    movel([0.080813, -1.351716, -2.594300, -0.766373, 1.570796, 1.651610],accel_mss,speed_ms,0,blend_radius_m)
    movel([0.080675, -1.351545, -2.594414, -0.766430, 1.570796, 1.651471],accel_mss,speed_ms,0,blend_radius_m)
    movel([0.080768, -1.351204, -2.594640, -0.766545, 1.570796, 1.651564],accel_mss,speed_ms,0,blend_radius_m)
    movel([0.080890, -1.350900, -2.594842, -0.766647, 1.570796, 1.651686],accel_mss,speed_ms,0,blend_radius_m)
    movel([0.080645, -1.350707, -2.594969, -0.766712, 1.570796, 1.651441],accel_mss,speed_ms,0,blend_radius_m)
    movel([0.080619, -1.350492, -2.595112, -0.766785, 1.570796, 1.651416],accel_mss,speed_ms,0,blend_radius_m)
    movel([0.080919, -1.350160, -2.595332, -0.766897, 1.570796, 1.651715],accel_mss,speed_ms,0,blend_radius_m)
    movel([0.080769, -1.349809, -2.595564, -0.767016, 1.570796, 1.651566],accel_mss,speed_ms,0,blend_radius_m)
    movel([0.080640, -1.349621, -2.595688, -0.767080, 1.570796, 1.651436],accel_mss,speed_ms,0,blend_radius_m)
    movel([0.080628, -1.349397, -2.595836, -0.767155, 1.570796, 1.651424],accel_mss,speed_ms,0,blend_radius_m)
    movel([0.080942, -1.348990, -2.596105, -0.767294, 1.570796, 1.651739],accel_mss,speed_ms,0,blend_radius_m)
    movel([0.081368, -1.348809, -2.596225, -0.767355, 1.570796, 1.652164],accel_mss,speed_ms,0,blend_radius_m)
    movel([0.083131, -1.348413, -2.596486, -0.767490, 1.570796, 1.653928],accel_mss,speed_ms,0,blend_radius_m)
    speed_ms = 0.003
    movel([0.083131, -1.335017, -2.590258, -0.787114, 1.570796, 1.653928],accel_mss,speed_ms,0,blend_radius_m)
    speed_ms = 1.000
    movel([0.083131, -1.309400, -2.577409, -0.825580, 1.570796, 1.653928],accel_mss,speed_ms,0,blend_radius_m)
    movel([0.082638, -1.312886, -2.575230, -0.824273, 1.570796, 1.653435],accel_mss,speed_ms,0,blend_radius_m)
    movel([0.082638, -1.338446, -2.588033, -0.785910, 1.570796, 1.653435],accel_mss,speed_ms,0,blend_radius_m)
    speed_ms = 0.003
    movel([0.082638, -1.348431, -2.592700, -0.771258, 1.570796, 1.653435],accel_mss,speed_ms,0,blend_radius_m)
    speed_ms = 0.007
    movel([0.083010, -1.348325, -2.592770, -0.771294, 1.570796, 1.653806],accel_mss,speed_ms,0,blend_radius_m)
    movel([0.083255, -1.348397, -2.592722, -0.771269, 1.570796, 1.654051],accel_mss,speed_ms,0,blend_radius_m)
    movel([0.083272, -1.348613, -2.592580, -0.771196, 1.570796, 1.654068],accel_mss,speed_ms,0,blend_radius_m)
    movel([0.082991, -1.348882, -2.592402, -0.771105, 1.570796, 1.653788],accel_mss,speed_ms,0,blend_radius_m)
    movel([0.082561, -1.349059, -2.592285, -0.771045, 1.570796, 1.653357],accel_mss,speed_ms,0,blend_radius_m)
    movel([0.082329, -1.349028, -2.592305, -0.771056, 1.570796, 1.653125],accel_mss,speed_ms,0,blend_radius_m)
    movel([0.082337, -1.348676, -2.592538, -0.771175, 1.570796, 1.653134],accel_mss,speed_ms,0,blend_radius_m)
    movel([0.082638, -1.348431, -2.592700, -0.771258, 1.570796, 1.653435],accel_mss,speed_ms,0,blend_radius_m)
    speed_ms = 0.003
    movel([0.082638, -1.351808, -2.594239, -0.766342, 1.570796, 1.653435],accel_mss,speed_ms,0,blend_radius_m)
    speed_ms = 0.007
    movel([0.083010, -1.351702, -2.594309, -0.766377, 1.570796, 1.653806],accel_mss,speed_ms,0,blend_radius_m)
    movel([0.083255, -1.351775, -2.594261, -0.766353, 1.570796, 1.654051],accel_mss,speed_ms,0,blend_radius_m)
    movel([0.083272, -1.351990, -2.594118, -0.766281, 1.570796, 1.654068],accel_mss,speed_ms,0,blend_radius_m)
    movel([0.082991, -1.352258, -2.593940, -0.766191, 1.570796, 1.653788],accel_mss,speed_ms,0,blend_radius_m)
    movel([0.082561, -1.352435, -2.593823, -0.766132, 1.570796, 1.653357],accel_mss,speed_ms,0,blend_radius_m)
    movel([0.082329, -1.352404, -2.593843, -0.766142, 1.570796, 1.653125],accel_mss,speed_ms,0,blend_radius_m)
    movel([0.082337, -1.352052, -2.594077, -0.766260, 1.570796, 1.653134],accel_mss,speed_ms,0,blend_radius_m)
    movel([0.082638, -1.351808, -2.594239, -0.766342, 1.570796, 1.653435],accel_mss,speed_ms,0,blend_radius_m)
    speed_ms = 0.003
    movel([0.082638, -1.338446, -2.588033, -0.785910, 1.570796, 1.653435],accel_mss,speed_ms,0,blend_radius_m)
    speed_ms = 1.000
    movel([0.082638, -1.312886, -2.575230, -0.824273, 1.570796, 1.653435],accel_mss,speed_ms,0,blend_radius_m)
    movel([0.075847, -1.319560, -2.571014, -0.821815, 1.570796, 1.646643],accel_mss,speed_ms,0,blend_radius_m)
    movel([0.075847, -1.345010, -2.583731, -0.783648, 1.570796, 1.646643],accel_mss,speed_ms,0,blend_radius_m)
    speed_ms = 0.003
    movel([0.075847, -1.354947, -2.588365, -0.769077, 1.570796, 1.646643],accel_mss,speed_ms,0,blend_radius_m)
    speed_ms = 0.007
    movel([0.076210, -1.355243, -2.588167, -0.768979, 1.570796, 1.647006],accel_mss,speed_ms,0,blend_radius_m)
    movel([0.076357, -1.355481, -2.588008, -0.768901, 1.570796, 1.647154],accel_mss,speed_ms,0,blend_radius_m)
    movel([0.076398, -1.355704, -2.587858, -0.768827, 1.570796, 1.647194],accel_mss,speed_ms,0,blend_radius_m)
    movel([0.076337, -1.355959, -2.587687, -0.768743, 1.570796, 1.647134],accel_mss,speed_ms,0,blend_radius_m)
    movel([0.076172, -1.356294, -2.587462, -0.768633, 1.570796, 1.646969],accel_mss,speed_ms,0,blend_radius_m)
    movel([0.075752, -1.356855, -2.587085, -0.768449, 1.570796, 1.646548],accel_mss,speed_ms,0,blend_radius_m)
    movel([0.075239, -1.357270, -2.586806, -0.768313, 1.570796, 1.646035],accel_mss,speed_ms,0,blend_radius_m)
    movel([0.074675, -1.357502, -2.586649, -0.768238, 1.570796, 1.645471],accel_mss,speed_ms,0,blend_radius_m)
    movel([0.074114, -1.357533, -2.586628, -0.768227, 1.570796, 1.644910],accel_mss,speed_ms,0,blend_radius_m)
    movel([0.073609, -1.357253, -2.586817, -0.768319, 1.570796, 1.644405],accel_mss,speed_ms,0,blend_radius_m)
    movel([0.073464, -1.356659, -2.587216, -0.768513, 1.570796, 1.644260],accel_mss,speed_ms,0,blend_radius_m)
    movel([0.073721, -1.355938, -2.587701, -0.768750, 1.570796, 1.644518],accel_mss,speed_ms,0,blend_radius_m)
    movel([0.074305, -1.355315, -2.588118, -0.768955, 1.570796, 1.645101],accel_mss,speed_ms,0,blend_radius_m)
    movel([0.074876, -1.354985, -2.588340, -0.769064, 1.570796, 1.645673],accel_mss,speed_ms,0,blend_radius_m)
    movel([0.075398, -1.354858, -2.588425, -0.769106, 1.570796, 1.646194],accel_mss,speed_ms,0,blend_radius_m)
    movel([0.075847, -1.354947, -2.588365, -0.769077, 1.570796, 1.646643],accel_mss,speed_ms,0,blend_radius_m)
    speed_ms = 0.003
    movel([0.075847, -1.358308, -2.589893, -0.764188, 1.570796, 1.646643],accel_mss,speed_ms,0,blend_radius_m)
    speed_ms = 0.007
    movel([0.076210, -1.358603, -2.589694, -0.764092, 1.570796, 1.647006],accel_mss,speed_ms,0,blend_radius_m)
    movel([0.076357, -1.358840, -2.589535, -0.764014, 1.570796, 1.647154],accel_mss,speed_ms,0,blend_radius_m)
    movel([0.076398, -1.359063, -2.589385, -0.763942, 1.570796, 1.647194],accel_mss,speed_ms,0,blend_radius_m)
    movel([0.076337, -1.359317, -2.589213, -0.763859, 1.570796, 1.647134],accel_mss,speed_ms,0,blend_radius_m)
    movel([0.076172, -1.359651, -2.588988, -0.763751, 1.570796, 1.646969],accel_mss,speed_ms,0,blend_radius_m)
    movel([0.075752, -1.360211, -2.588610, -0.763569, 1.570796, 1.646548],accel_mss,speed_ms,0,blend_radius_m)
    movel([0.075239, -1.360624, -2.588330, -0.763435, 1.570796, 1.646035],accel_mss,speed_ms,0,blend_radius_m)
    movel([0.074675, -1.360856, -2.588173, -0.763360, 1.570796, 1.645471],accel_mss,speed_ms,0,blend_radius_m)
    movel([0.074114, -1.360887, -2.588152, -0.763350, 1.570796, 1.644910],accel_mss,speed_ms,0,blend_radius_m)
    movel([0.073609, -1.360608, -2.588341, -0.763440, 1.570796, 1.644405],accel_mss,speed_ms,0,blend_radius_m)
    movel([0.073464, -1.360015, -2.588742, -0.763632, 1.570796, 1.644260],accel_mss,speed_ms,0,blend_radius_m)
    movel([0.073721, -1.359296, -2.589227, -0.763866, 1.570796, 1.644518],accel_mss,speed_ms,0,blend_radius_m)
    movel([0.074305, -1.358675, -2.589646, -0.764068, 1.570796, 1.645101],accel_mss,speed_ms,0,blend_radius_m)
    movel([0.074876, -1.358345, -2.589868, -0.764176, 1.570796, 1.645673],accel_mss,speed_ms,0,blend_radius_m)
    movel([0.075398, -1.358219, -2.589953, -0.764217, 1.570796, 1.646194],accel_mss,speed_ms,0,blend_radius_m)
    movel([0.075847, -1.358308, -2.589893, -0.764188, 1.570796, 1.646643],accel_mss,speed_ms,0,blend_radius_m)
    speed_ms = 0.003
    movel([0.075847, -1.345010, -2.583731, -0.783648, 1.570796, 1.646643],accel_mss,speed_ms,0,blend_radius_m)
    speed_ms = 1.000
    movel([0.075847, -1.319560, -2.571014, -0.821815, 1.570796, 1.646643],accel_mss,speed_ms,0,blend_radius_m)
    movel([0.078635, -1.323961, -2.568202, -0.820226, 1.570796, 1.649431],accel_mss,speed_ms,0,blend_radius_m)
    movel([0.078635, -1.349337, -2.580862, -0.782189, 1.570796, 1.649431],accel_mss,speed_ms,0,blend_radius_m)
    speed_ms = 0.003
    movel([0.078635, -1.359242, -2.585475, -0.767671, 1.570796, 1.649431],accel_mss,speed_ms,0,blend_radius_m)
    speed_ms = 0.007
    movel([0.079474, -1.359723, -2.585151, -0.767516, 1.570796, 1.650271],accel_mss,speed_ms,0,blend_radius_m)
    movel([0.080172, -1.360238, -2.584802, -0.767349, 1.570796, 1.650969],accel_mss,speed_ms,0,blend_radius_m)
    movel([0.080222, -1.360455, -2.584655, -0.767279, 1.570796, 1.651018],accel_mss,speed_ms,0,blend_radius_m)
    movel([0.079954, -1.360655, -2.584519, -0.767215, 1.570796, 1.650750],accel_mss,speed_ms,0,blend_radius_m)
    movel([0.079275, -1.360021, -2.584949, -0.767419, 1.570796, 1.650071],accel_mss,speed_ms,0,blend_radius_m)
    movel([0.078610, -1.359377, -2.585384, -0.767628, 1.570796, 1.649406],accel_mss,speed_ms,0,blend_radius_m)
    speed_ms = 0.003
    movel([0.078635, -1.362592, -2.586996, -0.762801, 1.570796, 1.649431],accel_mss,speed_ms,0,blend_radius_m)
    speed_ms = 0.007
    movel([0.079474, -1.363071, -2.586671, -0.762648, 1.570796, 1.650271],accel_mss,speed_ms,0,blend_radius_m)
    movel([0.080172, -1.363585, -2.586321, -0.762483, 1.570796, 1.650969],accel_mss,speed_ms,0,blend_radius_m)
    movel([0.080222, -1.363801, -2.586174, -0.762414, 1.570796, 1.651018],accel_mss,speed_ms,0,blend_radius_m)
    movel([0.079954, -1.364001, -2.586038, -0.762350, 1.570796, 1.650750],accel_mss,speed_ms,0,blend_radius_m)
    movel([0.079275, -1.363368, -2.586468, -0.762552, 1.570796, 1.650071],accel_mss,speed_ms,0,blend_radius_m)
    movel([0.078610, -1.362726, -2.586905, -0.762758, 1.570796, 1.649406],accel_mss,speed_ms,0,blend_radius_m)
    speed_ms = 0.003
    movel([0.078635, -1.349337, -2.580862, -0.782189, 1.570796, 1.649431],accel_mss,speed_ms,0,blend_radius_m)
    speed_ms = 1.000
    movel([0.078635, -1.323961, -2.568202, -0.820226, 1.570796, 1.649431],accel_mss,speed_ms,0,blend_radius_m)
    movel([0.084889, -1.331749, -2.563164, -0.817476, 1.570796, 1.655685],accel_mss,speed_ms,0,blend_radius_m)
    movel([0.084889, -1.356993, -2.575725, -0.779672, 1.570796, 1.655685],accel_mss,speed_ms,0,blend_radius_m)
    speed_ms = 0.003
    movel([0.084889, -1.366841, -2.580300, -0.765248, 1.570796, 1.655685],accel_mss,speed_ms,0,blend_radius_m)
    speed_ms = 0.007
    movel([0.085264, -1.366718, -2.580384, -0.765287, 1.570796, 1.656061],accel_mss,speed_ms,0,blend_radius_m)
    movel([0.085429, -1.367001, -2.580190, -0.765198, 1.570796, 1.656225],accel_mss,speed_ms,0,blend_radius_m)
    movel([0.085290, -1.367254, -2.580016, -0.765119, 1.570796, 1.656086],accel_mss,speed_ms,0,blend_radius_m)
    movel([0.085006, -1.367407, -2.579911, -0.765071, 1.570796, 1.655802],accel_mss,speed_ms,0,blend_radius_m)
    movel([0.084700, -1.367358, -2.579945, -0.765087, 1.570796, 1.655496],accel_mss,speed_ms,0,blend_radius_m)
    movel([0.084687, -1.367140, -2.580094, -0.765155, 1.570796, 1.655483],accel_mss,speed_ms,0,blend_radius_m)
    movel([0.084889, -1.366841, -2.580300, -0.765248, 1.570796, 1.655685],accel_mss,speed_ms,0,blend_radius_m)
    speed_ms = 0.003
    movel([0.084889, -1.370170, -2.581808, -0.760411, 1.570796, 1.655685],accel_mss,speed_ms,0,blend_radius_m)
    speed_ms = 0.007
    movel([0.085264, -1.370048, -2.581893, -0.760449, 1.570796, 1.656061],accel_mss,speed_ms,0,blend_radius_m)
    movel([0.085429, -1.370330, -2.581698, -0.760361, 1.570796, 1.656225],accel_mss,speed_ms,0,blend_radius_m)
    movel([0.085290, -1.370582, -2.581524, -0.760283, 1.570796, 1.656086],accel_mss,speed_ms,0,blend_radius_m)
    movel([0.085006, -1.370735, -2.581418, -0.760236, 1.570796, 1.655802],accel_mss,speed_ms,0,blend_radius_m)
    movel([0.084700, -1.370686, -2.581452, -0.760251, 1.570796, 1.655496],accel_mss,speed_ms,0,blend_radius_m)
    movel([0.084687, -1.370469, -2.581602, -0.760318, 1.570796, 1.655483],accel_mss,speed_ms,0,blend_radius_m)
    movel([0.084889, -1.370170, -2.581808, -0.760411, 1.570796, 1.655685],accel_mss,speed_ms,0,blend_radius_m)
    speed_ms = 0.003
    movel([0.084889, -1.356993, -2.575725, -0.779672, 1.570796, 1.655685],accel_mss,speed_ms,0,blend_radius_m)
    speed_ms = 1.000
    movel([0.084889, -1.331749, -2.563164, -0.817476, 1.570796, 1.655685],accel_mss,speed_ms,0,blend_radius_m)
    movel([0.086824, -1.329871, -2.564386, -0.818131, 1.570796, 1.657620],accel_mss,speed_ms,0,blend_radius_m)
    movel([0.086824, -1.355147, -2.576970, -0.780271, 1.570796, 1.657620],accel_mss,speed_ms,0,blend_radius_m)
    speed_ms = 0.003
    movel([0.086824, -1.365009, -2.581555, -0.765825, 1.570796, 1.657620],accel_mss,speed_ms,0,blend_radius_m)
    speed_ms = 0.007
    movel([0.087168, -1.365279, -2.581370, -0.765740, 1.570796, 1.657964],accel_mss,speed_ms,0,blend_radius_m)
    movel([0.087391, -1.365516, -2.581208, -0.765665, 1.570796, 1.658187],accel_mss,speed_ms,0,blend_radius_m)
    movel([0.087551, -1.365788, -2.581021, -0.765579, 1.570796, 1.658347],accel_mss,speed_ms,0,blend_radius_m)
    movel([0.087693, -1.366165, -2.580764, -0.765461, 1.570796, 1.658489],accel_mss,speed_ms,0,blend_radius_m)
    movel([0.087762, -1.366699, -2.580397, -0.765293, 1.570796, 1.658558],accel_mss,speed_ms,0,blend_radius_m)
    movel([0.087686, -1.367444, -2.579885, -0.765060, 1.570796, 1.658482],accel_mss,speed_ms,0,blend_radius_m)
    movel([0.087505, -1.368211, -2.579358, -0.764820, 1.570796, 1.658301],accel_mss,speed_ms,0,blend_radius_m)
    movel([0.087241, -1.368817, -2.578940, -0.764632, 1.570796, 1.658038],accel_mss,speed_ms,0,blend_radius_m)
    movel([0.086827, -1.369458, -2.578498, -0.764433, 1.570796, 1.657623],accel_mss,speed_ms,0,blend_radius_m)
    movel([0.086336, -1.370058, -2.578084, -0.764247, 1.570796, 1.657133],accel_mss,speed_ms,0,blend_radius_m)
    movel([0.085769, -1.370615, -2.577699, -0.764075, 1.570796, 1.656565],accel_mss,speed_ms,0,blend_radius_m)
    movel([0.085120, -1.371138, -2.577337, -0.763914, 1.570796, 1.655916],accel_mss,speed_ms,0,blend_radius_m)
    movel([0.084603, -1.371499, -2.577086, -0.763803, 1.570796, 1.655399],accel_mss,speed_ms,0,blend_radius_m)
    movel([0.084238, -1.371707, -2.576942, -0.763740, 1.570796, 1.655035],accel_mss,speed_ms,0,blend_radius_m)
    movel([0.083834, -1.371872, -2.576828, -0.763689, 1.570796, 1.654631],accel_mss,speed_ms,0,blend_radius_m)
    movel([0.083145, -1.372087, -2.576679, -0.763623, 1.570796, 1.653941],accel_mss,speed_ms,0,blend_radius_m)
    movel([0.082486, -1.372273, -2.576550, -0.763566, 1.570796, 1.653282],accel_mss,speed_ms,0,blend_radius_m)
    movel([0.082081, -1.372352, -2.576495, -0.763542, 1.570796, 1.652877],accel_mss,speed_ms,0,blend_radius_m)
    movel([0.081735, -1.372366, -2.576485, -0.763538, 1.570796, 1.652532],accel_mss,speed_ms,0,blend_radius_m)
    movel([0.081304, -1.372326, -2.576513, -0.763550, 1.570796, 1.652101],accel_mss,speed_ms,0,blend_radius_m)
    movel([0.080718, -1.372180, -2.576614, -0.763595, 1.570796, 1.651515],accel_mss,speed_ms,0,blend_radius_m)
    movel([0.080185, -1.371922, -2.576793, -0.763674, 1.570796, 1.650981],accel_mss,speed_ms,0,blend_radius_m)
    movel([0.079747, -1.371571, -2.577037, -0.763781, 1.570796, 1.650544],accel_mss,speed_ms,0,blend_radius_m)
    movel([0.079442, -1.371152, -2.577327, -0.763910, 1.570796, 1.650238],accel_mss,speed_ms,0,blend_radius_m)
    movel([0.079335, -1.370890, -2.577508, -0.763991, 1.570796, 1.650132],accel_mss,speed_ms,0,blend_radius_m)
    movel([0.079280, -1.370612, -2.577701, -0.764076, 1.570796, 1.650076],accel_mss,speed_ms,0,blend_radius_m)
    movel([0.079271, -1.370257, -2.577947, -0.764186, 1.570796, 1.650067],accel_mss,speed_ms,0,blend_radius_m)
    movel([0.079306, -1.369743, -2.578301, -0.764344, 1.570796, 1.650102],accel_mss,speed_ms,0,blend_radius_m)
    movel([0.079370, -1.369178, -2.578691, -0.764520, 1.570796, 1.650167],accel_mss,speed_ms,0,blend_radius_m)
    movel([0.079452, -1.368805, -2.578949, -0.764635, 1.570796, 1.650248],accel_mss,speed_ms,0,blend_radius_m)
    movel([0.079585, -1.368463, -2.579184, -0.764742, 1.570796, 1.650381],accel_mss,speed_ms,0,blend_radius_m)
    movel([0.079810, -1.368029, -2.579483, -0.764877, 1.570796, 1.650606],accel_mss,speed_ms,0,blend_radius_m)
    movel([0.080321, -1.367272, -2.580004, -0.765113, 1.570796, 1.651117],accel_mss,speed_ms,0,blend_radius_m)
    movel([0.080995, -1.366513, -2.580524, -0.765351, 1.570796, 1.651792],accel_mss,speed_ms,0,blend_radius_m)
    movel([0.081741, -1.365848, -2.580980, -0.765560, 1.570796, 1.652537],accel_mss,speed_ms,0,blend_radius_m)
    movel([0.082465, -1.365369, -2.581309, -0.765711, 1.570796, 1.653262],accel_mss,speed_ms,0,blend_radius_m)
    movel([0.083702, -1.364840, -2.581671, -0.765879, 1.570796, 1.654499],accel_mss,speed_ms,0,blend_radius_m)
    movel([0.084908, -1.364595, -2.581838, -0.765956, 1.570796, 1.655704],accel_mss,speed_ms,0,blend_radius_m)
    movel([0.085979, -1.364652, -2.581799, -0.765938, 1.570796, 1.656775],accel_mss,speed_ms,0,blend_radius_m)
    movel([0.086824, -1.365009, -2.581555, -0.765825, 1.570796, 1.657620],accel_mss,speed_ms,0,blend_radius_m)
    speed_ms = 0.003
    movel([0.086824, -1.368344, -2.583066, -0.760979, 1.570796, 1.657620],accel_mss,speed_ms,0,blend_radius_m)
    speed_ms = 0.007
    movel([0.087168, -1.368612, -2.582881, -0.760896, 1.570796, 1.657964],accel_mss,speed_ms,0,blend_radius_m)
    movel([0.087391, -1.368849, -2.582719, -0.760822, 1.570796, 1.658187],accel_mss,speed_ms,0,blend_radius_m)
    movel([0.087551, -1.369121, -2.582531, -0.760737, 1.570796, 1.658347],accel_mss,speed_ms,0,blend_radius_m)
    movel([0.087693, -1.369496, -2.582273, -0.760620, 1.570796, 1.658489],accel_mss,speed_ms,0,blend_radius_m)
    movel([0.087762, -1.370029, -2.581906, -0.760455, 1.570796, 1.658558],accel_mss,speed_ms,0,blend_radius_m)
    movel([0.087686, -1.370772, -2.581393, -0.760224, 1.570796, 1.658482],accel_mss,speed_ms,0,blend_radius_m)
    movel([0.087505, -1.371537, -2.580864, -0.759988, 1.570796, 1.658301],accel_mss,speed_ms,0,blend_radius_m)
    movel([0.087241, -1.372141, -2.580445, -0.759802, 1.570796, 1.658038],accel_mss,speed_ms,0,blend_radius_m)
    movel([0.086827, -1.372781, -2.580002, -0.759606, 1.570796, 1.657623],accel_mss,speed_ms,0,blend_radius_m)
    movel([0.086336, -1.373379, -2.579587, -0.759423, 1.570796, 1.657133],accel_mss,speed_ms,0,blend_radius_m)
    movel([0.085769, -1.373934, -2.579201, -0.759254, 1.570796, 1.656565],accel_mss,speed_ms,0,blend_radius_m)
    movel([0.085120, -1.374456, -2.578838, -0.759095, 1.570796, 1.655916],accel_mss,speed_ms,0,blend_radius_m)
    movel([0.084603, -1.374816, -2.578587, -0.758986, 1.570796, 1.655399],accel_mss,speed_ms,0,blend_radius_m)
    movel([0.084238, -1.375023, -2.578443, -0.758923, 1.570796, 1.655035],accel_mss,speed_ms,0,blend_radius_m)
    movel([0.083834, -1.375188, -2.578328, -0.758873, 1.570796, 1.654631],accel_mss,speed_ms,0,blend_radius_m)
    movel([0.083145, -1.375403, -2.578178, -0.758808, 1.570796, 1.653941],accel_mss,speed_ms,0,blend_radius_m)
    movel([0.082486, -1.375588, -2.578049, -0.758752, 1.570796, 1.653282],accel_mss,speed_ms,0,blend_radius_m)
    movel([0.082081, -1.375667, -2.577994, -0.758728, 1.570796, 1.652877],accel_mss,speed_ms,0,blend_radius_m)
    movel([0.081735, -1.375681, -2.577984, -0.758724, 1.570796, 1.652532],accel_mss,speed_ms,0,blend_radius_m)
    movel([0.081304, -1.375641, -2.578012, -0.758736, 1.570796, 1.652101],accel_mss,speed_ms,0,blend_radius_m)
    movel([0.080718, -1.375495, -2.578114, -0.758780, 1.570796, 1.651515],accel_mss,speed_ms,0,blend_radius_m)
    movel([0.080185, -1.375238, -2.578293, -0.758858, 1.570796, 1.650981],accel_mss,speed_ms,0,blend_radius_m)
    movel([0.079747, -1.374887, -2.578537, -0.758964, 1.570796, 1.650544],accel_mss,speed_ms,0,blend_radius_m)
    movel([0.079442, -1.374470, -2.578828, -0.759091, 1.570796, 1.650238],accel_mss,speed_ms,0,blend_radius_m)
    movel([0.079335, -1.374209, -2.579010, -0.759170, 1.570796, 1.650132],accel_mss,speed_ms,0,blend_radius_m)
    movel([0.079280, -1.373932, -2.579203, -0.759255, 1.570796, 1.650076],accel_mss,speed_ms,0,blend_radius_m)
    movel([0.079271, -1.373577, -2.579449, -0.759363, 1.570796, 1.650067],accel_mss,speed_ms,0,blend_radius_m)
    movel([0.079306, -1.373065, -2.579805, -0.759519, 1.570796, 1.650102],accel_mss,speed_ms,0,blend_radius_m)
    movel([0.079370, -1.372501, -2.580196, -0.759692, 1.570796, 1.650167],accel_mss,speed_ms,0,blend_radius_m)
    movel([0.079452, -1.372129, -2.580454, -0.759806, 1.570796, 1.650248],accel_mss,speed_ms,0,blend_radius_m)
    movel([0.079585, -1.371788, -2.580690, -0.759911, 1.570796, 1.650381],accel_mss,speed_ms,0,blend_radius_m)
    movel([0.079810, -1.371355, -2.580990, -0.760044, 1.570796, 1.650606],accel_mss,speed_ms,0,blend_radius_m)
    movel([0.080321, -1.370600, -2.581511, -0.760278, 1.570796, 1.651117],accel_mss,speed_ms,0,blend_radius_m)
    movel([0.080995, -1.369844, -2.582033, -0.760512, 1.570796, 1.651792],accel_mss,speed_ms,0,blend_radius_m)
    movel([0.081741, -1.369180, -2.582490, -0.760718, 1.570796, 1.652537],accel_mss,speed_ms,0,blend_radius_m)
    movel([0.082465, -1.368702, -2.582819, -0.760867, 1.570796, 1.653262],accel_mss,speed_ms,0,blend_radius_m)
    movel([0.083702, -1.368175, -2.583182, -0.761032, 1.570796, 1.654499],accel_mss,speed_ms,0,blend_radius_m)
    movel([0.084908, -1.367930, -2.583350, -0.761109, 1.570796, 1.655704],accel_mss,speed_ms,0,blend_radius_m)
    movel([0.085979, -1.367988, -2.583311, -0.761091, 1.570796, 1.656775],accel_mss,speed_ms,0,blend_radius_m)
    movel([0.086824, -1.368344, -2.583066, -0.760979, 1.570796, 1.657620],accel_mss,speed_ms,0,blend_radius_m)
    speed_ms = 0.003
    movel([0.086824, -1.355147, -2.576970, -0.780271, 1.570796, 1.657620],accel_mss,speed_ms,0,blend_radius_m)
    speed_ms = 1.000
    movel([0.086824, -1.329871, -2.564386, -0.818131, 1.570796, 1.657620],accel_mss,speed_ms,0,blend_radius_m)
    movel([0.094772, -1.328855, -2.565045, -0.818488, 1.570796, 1.665569],accel_mss,speed_ms,0,blend_radius_m)
    movel([0.094772, -1.354149, -2.577643, -0.780598, 1.570796, 1.665569],accel_mss,speed_ms,0,blend_radius_m)
    speed_ms = 0.003
    movel([0.094772, -1.364018, -2.582232, -0.766139, 1.570796, 1.665569],accel_mss,speed_ms,0,blend_radius_m)
    speed_ms = 0.007
    movel([0.094995, -1.363677, -2.582465, -0.766248, 1.570796, 1.665791],accel_mss,speed_ms,0,blend_radius_m)
    movel([0.095323, -1.363701, -2.582448, -0.766240, 1.570796, 1.666120],accel_mss,speed_ms,0,blend_radius_m)
    movel([0.095419, -1.363975, -2.582261, -0.766153, 1.570796, 1.666215],accel_mss,speed_ms,0,blend_radius_m)
    movel([0.095125, -1.364292, -2.582045, -0.766052, 1.570796, 1.665921],accel_mss,speed_ms,0,blend_radius_m)
    movel([0.094811, -1.364341, -2.582011, -0.766037, 1.570796, 1.665607],accel_mss,speed_ms,0,blend_radius_m)
    movel([0.094772, -1.364018, -2.582232, -0.766139, 1.570796, 1.665569],accel_mss,speed_ms,0,blend_radius_m)
    speed_ms = 0.003
    movel([0.094772, -1.367355, -2.583745, -0.761289, 1.570796, 1.665569],accel_mss,speed_ms,0,blend_radius_m)
    speed_ms = 0.007
    movel([0.094995, -1.367014, -2.583978, -0.761396, 1.570796, 1.665791],accel_mss,speed_ms,0,blend_radius_m)
    movel([0.095323, -1.367038, -2.583962, -0.761389, 1.570796, 1.666120],accel_mss,speed_ms,0,blend_radius_m)
    movel([0.095419, -1.367312, -2.583774, -0.761303, 1.570796, 1.666215],accel_mss,speed_ms,0,blend_radius_m)
    movel([0.095125, -1.367628, -2.583557, -0.761203, 1.570796, 1.665921],accel_mss,speed_ms,0,blend_radius_m)
    movel([0.094811, -1.367677, -2.583524, -0.761188, 1.570796, 1.665607],accel_mss,speed_ms,0,blend_radius_m)
    movel([0.094772, -1.367355, -2.583745, -0.761289, 1.570796, 1.665569],accel_mss,speed_ms,0,blend_radius_m)
    speed_ms = 0.003
    movel([0.094772, -1.354149, -2.577643, -0.780598, 1.570796, 1.665569],accel_mss,speed_ms,0,blend_radius_m)
    speed_ms = 1.000
    movel([0.094772, -1.328855, -2.565045, -0.818488, 1.570796, 1.665569],accel_mss,speed_ms,0,blend_radius_m)
    movel([0.093044, -1.328349, -2.565373, -0.818667, 1.570796, 1.663841],accel_mss,speed_ms,0,blend_radius_m)
    movel([0.093044, -1.353651, -2.577977, -0.780761, 1.570796, 1.663841],accel_mss,speed_ms,0,blend_radius_m)
    speed_ms = 0.003
    movel([0.093044, -1.363524, -2.582569, -0.766296, 1.570796, 1.663841],accel_mss,speed_ms,0,blend_radius_m)
    speed_ms = 0.007
    movel([0.093644, -1.362822, -2.583047, -0.766520, 1.570796, 1.664441],accel_mss,speed_ms,0,blend_radius_m)
    movel([0.094331, -1.362169, -2.583491, -0.766728, 1.570796, 1.665128],accel_mss,speed_ms,0,blend_radius_m)
    movel([0.095046, -1.361633, -2.583856, -0.766900, 1.570796, 1.665842],accel_mss,speed_ms,0,blend_radius_m)
    movel([0.096773, -1.360824, -2.584405, -0.767160, 1.570796, 1.667569],accel_mss,speed_ms,0,blend_radius_m)
    movel([0.098461, -1.360629, -2.584537, -0.767223, 1.570796, 1.669258],accel_mss,speed_ms,0,blend_radius_m)
    movel([0.099813, -1.361083, -2.584229, -0.767077, 1.570796, 1.670609],accel_mss,speed_ms,0,blend_radius_m)
    movel([0.100589, -1.362108, -2.583533, -0.766748, 1.570796, 1.671385],accel_mss,speed_ms,0,blend_radius_m)
    movel([0.100651, -1.362593, -2.583203, -0.766593, 1.570796, 1.671448],accel_mss,speed_ms,0,blend_radius_m)
    movel([0.100652, -1.362928, -2.582975, -0.766486, 1.570796, 1.671448],accel_mss,speed_ms,0,blend_radius_m)
    movel([0.100628, -1.363261, -2.582748, -0.766380, 1.570796, 1.671424],accel_mss,speed_ms,0,blend_radius_m)
    movel([0.100362, -1.364362, -2.581997, -0.766030, 1.570796, 1.671159],accel_mss,speed_ms,0,blend_radius_m)
    movel([0.099808, -1.365429, -2.581267, -0.765692, 1.570796, 1.670604],accel_mss,speed_ms,0,blend_radius_m)
    movel([0.098981, -1.366422, -2.580587, -0.765380, 1.570796, 1.669777],accel_mss,speed_ms,0,blend_radius_m)
    movel([0.097911, -1.367310, -2.579977, -0.765101, 1.570796, 1.668707],accel_mss,speed_ms,0,blend_radius_m)
    movel([0.097420, -1.367637, -2.579752, -0.764999, 1.570796, 1.668216],accel_mss,speed_ms,0,blend_radius_m)
    movel([0.097050, -1.367840, -2.579613, -0.764936, 1.570796, 1.667847],accel_mss,speed_ms,0,blend_radius_m)
    movel([0.096644, -1.368002, -2.579502, -0.764885, 1.570796, 1.667440],accel_mss,speed_ms,0,blend_radius_m)
    movel([0.096013, -1.368199, -2.579366, -0.764824, 1.570796, 1.666809],accel_mss,speed_ms,0,blend_radius_m)
    movel([0.095377, -1.368373, -2.579247, -0.764770, 1.570796, 1.666173],accel_mss,speed_ms,0,blend_radius_m)
    movel([0.094976, -1.368446, -2.579196, -0.764747, 1.570796, 1.665772],accel_mss,speed_ms,0,blend_radius_m)
    movel([0.094614, -1.368453, -2.579191, -0.764745, 1.570796, 1.665410],accel_mss,speed_ms,0,blend_radius_m)
    movel([0.094128, -1.368401, -2.579227, -0.764761, 1.570796, 1.664925],accel_mss,speed_ms,0,blend_radius_m)
    movel([0.093507, -1.368260, -2.579324, -0.764805, 1.570796, 1.664303],accel_mss,speed_ms,0,blend_radius_m)
    movel([0.093023, -1.368028, -2.579484, -0.764877, 1.570796, 1.663819],accel_mss,speed_ms,0,blend_radius_m)
    movel([0.092642, -1.367684, -2.579721, -0.764985, 1.570796, 1.663438],accel_mss,speed_ms,0,blend_radius_m)
    movel([0.092324, -1.367203, -2.580051, -0.765135, 1.570796, 1.663120],accel_mss,speed_ms,0,blend_radius_m)
    movel([0.092145, -1.366594, -2.580469, -0.765326, 1.570796, 1.662941],accel_mss,speed_ms,0,blend_radius_m)
    movel([0.092139, -1.365795, -2.581017, -0.765577, 1.570796, 1.662936],accel_mss,speed_ms,0,blend_radius_m)
    movel([0.092293, -1.364952, -2.581594, -0.765843, 1.570796, 1.663090],accel_mss,speed_ms,0,blend_radius_m)
    movel([0.092597, -1.364210, -2.582101, -0.766078, 1.570796, 1.663394],accel_mss,speed_ms,0,blend_radius_m)
    movel([0.093044, -1.363524, -2.582569, -0.766296, 1.570796, 1.663841],accel_mss,speed_ms,0,blend_radius_m)
    speed_ms = 0.003
    movel([0.093044, -1.366862, -2.584083, -0.761444, 1.570796, 1.663841],accel_mss,speed_ms,0,blend_radius_m)
    speed_ms = 0.007
    movel([0.093644, -1.366162, -2.584562, -0.761665, 1.570796, 1.664441],accel_mss,speed_ms,0,blend_radius_m)
    movel([0.094331, -1.365511, -2.585007, -0.761871, 1.570796, 1.665128],accel_mss,speed_ms,0,blend_radius_m)
    movel([0.095046, -1.364976, -2.585373, -0.762040, 1.570796, 1.665842],accel_mss,speed_ms,0,blend_radius_m)
    movel([0.096773, -1.364169, -2.585923, -0.762297, 1.570796, 1.667569],accel_mss,speed_ms,0,blend_radius_m)
    movel([0.098461, -1.363974, -2.586056, -0.762359, 1.570796, 1.669258],accel_mss,speed_ms,0,blend_radius_m)
    movel([0.099813, -1.364427, -2.585747, -0.762215, 1.570796, 1.670609],accel_mss,speed_ms,0,blend_radius_m)
    movel([0.100589, -1.365450, -2.585049, -0.761890, 1.570796, 1.671385],accel_mss,speed_ms,0,blend_radius_m)
    movel([0.100651, -1.365933, -2.584718, -0.761737, 1.570796, 1.671448],accel_mss,speed_ms,0,blend_radius_m)
    movel([0.100652, -1.366267, -2.584490, -0.761632, 1.570796, 1.671448],accel_mss,speed_ms,0,blend_radius_m)
    movel([0.100628, -1.366600, -2.584262, -0.761527, 1.570796, 1.671424],accel_mss,speed_ms,0,blend_radius_m)
    movel([0.100362, -1.367698, -2.583509, -0.761181, 1.570796, 1.671159],accel_mss,speed_ms,0,blend_radius_m)
    movel([0.099808, -1.368763, -2.582778, -0.760849, 1.570796, 1.670604],accel_mss,speed_ms,0,blend_radius_m)
    movel([0.098981, -1.369752, -2.582096, -0.760540, 1.570796, 1.669777],accel_mss,speed_ms,0,blend_radius_m)
    movel([0.097911, -1.370638, -2.581485, -0.760266, 1.570796, 1.668707],accel_mss,speed_ms,0,blend_radius_m)
    movel([0.097420, -1.370965, -2.581259, -0.760165, 1.570796, 1.668216],accel_mss,speed_ms,0,blend_radius_m)
    movel([0.097050, -1.371167, -2.581120, -0.760103, 1.570796, 1.667847],accel_mss,speed_ms,0,blend_radius_m)
    movel([0.096644, -1.371328, -2.581008, -0.760053, 1.570796, 1.667440],accel_mss,speed_ms,0,blend_radius_m)
    movel([0.096013, -1.371525, -2.580872, -0.759992, 1.570796, 1.666809],accel_mss,speed_ms,0,blend_radius_m)
    movel([0.095377, -1.371698, -2.580752, -0.759939, 1.570796, 1.666173],accel_mss,speed_ms,0,blend_radius_m)
    movel([0.094976, -1.371771, -2.580701, -0.759916, 1.570796, 1.665772],accel_mss,speed_ms,0,blend_radius_m)
    movel([0.094614, -1.371778, -2.580697, -0.759914, 1.570796, 1.665410],accel_mss,speed_ms,0,blend_radius_m)
    movel([0.094128, -1.371726, -2.580733, -0.759930, 1.570796, 1.664925],accel_mss,speed_ms,0,blend_radius_m)
    movel([0.093507, -1.371585, -2.580830, -0.759973, 1.570796, 1.664303],accel_mss,speed_ms,0,blend_radius_m)
    movel([0.093023, -1.371354, -2.580990, -0.760045, 1.570796, 1.663819],accel_mss,speed_ms,0,blend_radius_m)
    movel([0.092642, -1.371011, -2.581228, -0.760151, 1.570796, 1.663438],accel_mss,speed_ms,0,blend_radius_m)
    movel([0.092324, -1.370532, -2.581559, -0.760299, 1.570796, 1.663120],accel_mss,speed_ms,0,blend_radius_m)
    movel([0.092145, -1.369924, -2.581978, -0.760487, 1.570796, 1.662941],accel_mss,speed_ms,0,blend_radius_m)
    movel([0.092139, -1.369127, -2.582527, -0.760735, 1.570796, 1.662936],accel_mss,speed_ms,0,blend_radius_m)
    movel([0.092293, -1.368287, -2.583105, -0.760997, 1.570796, 1.663090],accel_mss,speed_ms,0,blend_radius_m)
    movel([0.092597, -1.367547, -2.583613, -0.761229, 1.570796, 1.663394],accel_mss,speed_ms,0,blend_radius_m)
    movel([0.093044, -1.366862, -2.584083, -0.761444, 1.570796, 1.663841],accel_mss,speed_ms,0,blend_radius_m)
    speed_ms = 0.003
    movel([0.093044, -1.353651, -2.577977, -0.780761, 1.570796, 1.663841],accel_mss,speed_ms,0,blend_radius_m)
    speed_ms = 1.000
    movel([0.093044, -1.328349, -2.565373, -0.818667, 1.570796, 1.663841],accel_mss,speed_ms,0,blend_radius_m)
    movel([0.093095, -1.337880, -2.559143, -0.815367, 1.570796, 1.663891],accel_mss,speed_ms,0,blend_radius_m)
    movel([0.093095, -1.363017, -2.571624, -0.777747, 1.570796, 1.663891],accel_mss,speed_ms,0,blend_radius_m)
    speed_ms = 0.003
    movel([0.093095, -1.372820, -2.576170, -0.763399, 1.570796, 1.663891],accel_mss,speed_ms,0,blend_radius_m)
    speed_ms = 0.007
    movel([0.095667, -1.371889, -2.576816, -0.763684, 1.570796, 1.666464],accel_mss,speed_ms,0,blend_radius_m)
    movel([0.097439, -1.371146, -2.577331, -0.763912, 1.570796, 1.668235],accel_mss,speed_ms,0,blend_radius_m)
    movel([0.099151, -1.370361, -2.577874, -0.764154, 1.570796, 1.669947],accel_mss,speed_ms,0,blend_radius_m)
    movel([0.100738, -1.369566, -2.578424, -0.764399, 1.570796, 1.671535],accel_mss,speed_ms,0,blend_radius_m)
    movel([0.102129, -1.368796, -2.578955, -0.764638, 1.570796, 1.672925],accel_mss,speed_ms,0,blend_radius_m)
    movel([0.103079, -1.368244, -2.579335, -0.764810, 1.570796, 1.673875],accel_mss,speed_ms,0,blend_radius_m)
    movel([0.103407, -1.368085, -2.579445, -0.764859, 1.570796, 1.674203],accel_mss,speed_ms,0,blend_radius_m)
    movel([0.103782, -1.368141, -2.579406, -0.764842, 1.570796, 1.674579],accel_mss,speed_ms,0,blend_radius_m)
    movel([0.103972, -1.368477, -2.579175, -0.764737, 1.570796, 1.674769],accel_mss,speed_ms,0,blend_radius_m)
    movel([0.104047, -1.369268, -2.578630, -0.764492, 1.570796, 1.674843],accel_mss,speed_ms,0,blend_radius_m)
    movel([0.104025, -1.370097, -2.578057, -0.764235, 1.570796, 1.674822],accel_mss,speed_ms,0,blend_radius_m)
    movel([0.103868, -1.370632, -2.577687, -0.764070, 1.570796, 1.674664],accel_mss,speed_ms,0,blend_radius_m)
    movel([0.103307, -1.371174, -2.577312, -0.763903, 1.570796, 1.674104],accel_mss,speed_ms,0,blend_radius_m)
    movel([0.100371, -1.372580, -2.576336, -0.763472, 1.570796, 1.671167],accel_mss,speed_ms,0,blend_radius_m)
    movel([0.097202, -1.373985, -2.575359, -0.763045, 1.570796, 1.667998],accel_mss,speed_ms,0,blend_radius_m)
    movel([0.094275, -1.375126, -2.574563, -0.762700, 1.570796, 1.665072],accel_mss,speed_ms,0,blend_radius_m)
    movel([0.091963, -1.375881, -2.574036, -0.762472, 1.570796, 1.662759],accel_mss,speed_ms,0,blend_radius_m)
    movel([0.088651, -1.376817, -2.573380, -0.762191, 1.570796, 1.659447],accel_mss,speed_ms,0,blend_radius_m)
    movel([0.085300, -1.377694, -2.572766, -0.761930, 1.570796, 1.656096],accel_mss,speed_ms,0,blend_radius_m)
    movel([0.082794, -1.378255, -2.572372, -0.761763, 1.570796, 1.653590],accel_mss,speed_ms,0,blend_radius_m)
    movel([0.080908, -1.378590, -2.572136, -0.761663, 1.570796, 1.651704],accel_mss,speed_ms,0,blend_radius_m)
    movel([0.078698, -1.378923, -2.571902, -0.761564, 1.570796, 1.649495],accel_mss,speed_ms,0,blend_radius_m)
    movel([0.076615, -1.379200, -2.571707, -0.761482, 1.570796, 1.647412],accel_mss,speed_ms,0,blend_radius_m)
    movel([0.075933, -1.379208, -2.571701, -0.761480, 1.570796, 1.646730],accel_mss,speed_ms,0,blend_radius_m)
    movel([0.075687, -1.379042, -2.571818, -0.761529, 1.570796, 1.646483],accel_mss,speed_ms,0,blend_radius_m)
    movel([0.075673, -1.378811, -2.571981, -0.761597, 1.570796, 1.646469],accel_mss,speed_ms,0,blend_radius_m)
    movel([0.075722, -1.378205, -2.572406, -0.761777, 1.570796, 1.646518],accel_mss,speed_ms,0,blend_radius_m)
    movel([0.075826, -1.377463, -2.572928, -0.761998, 1.570796, 1.646623],accel_mss,speed_ms,0,blend_radius_m)
    movel([0.075986, -1.376875, -2.573340, -0.762174, 1.570796, 1.646783],accel_mss,speed_ms,0,blend_radius_m)
    movel([0.076193, -1.376445, -2.573641, -0.762303, 1.570796, 1.646990],accel_mss,speed_ms,0,blend_radius_m)
    movel([0.076445, -1.376205, -2.573809, -0.762375, 1.570796, 1.647241],accel_mss,speed_ms,0,blend_radius_m)
    movel([0.076934, -1.376110, -2.573875, -0.762403, 1.570796, 1.647730],accel_mss,speed_ms,0,blend_radius_m)
    movel([0.077336, -1.376082, -2.573895, -0.762412, 1.570796, 1.648132],accel_mss,speed_ms,0,blend_radius_m)
    movel([0.077768, -1.376072, -2.573902, -0.762415, 1.570796, 1.648564],accel_mss,speed_ms,0,blend_radius_m)
    movel([0.078966, -1.376038, -2.573926, -0.762425, 1.570796, 1.649762],accel_mss,speed_ms,0,blend_radius_m)
    movel([0.080402, -1.375921, -2.574008, -0.762460, 1.570796, 1.651198],accel_mss,speed_ms,0,blend_radius_m)
    movel([0.081934, -1.375738, -2.574136, -0.762515, 1.570796, 1.652730],accel_mss,speed_ms,0,blend_radius_m)
    movel([0.083427, -1.375504, -2.574300, -0.762586, 1.570796, 1.654223],accel_mss,speed_ms,0,blend_radius_m)
    movel([0.085813, -1.374972, -2.574671, -0.762746, 1.570796, 1.656609],accel_mss,speed_ms,0,blend_radius_m)
    movel([0.089434, -1.373949, -2.575384, -0.763056, 1.570796, 1.660230],accel_mss,speed_ms,0,blend_radius_m)
    movel([0.093095, -1.372820, -2.576170, -0.763399, 1.570796, 1.663891],accel_mss,speed_ms,0,blend_radius_m)
    speed_ms = 0.003
    movel([0.093095, -1.376133, -2.577668, -0.758587, 1.570796, 1.663891],accel_mss,speed_ms,0,blend_radius_m)
    speed_ms = 0.007
    movel([0.095667, -1.375205, -2.578316, -0.758868, 1.570796, 1.666464],accel_mss,speed_ms,0,blend_radius_m)
    movel([0.097439, -1.374463, -2.578833, -0.759093, 1.570796, 1.668235],accel_mss,speed_ms,0,blend_radius_m)
    movel([0.099151, -1.373681, -2.579377, -0.759331, 1.570796, 1.669947],accel_mss,speed_ms,0,blend_radius_m)
    movel([0.100738, -1.372888, -2.579927, -0.759573, 1.570796, 1.671535],accel_mss,speed_ms,0,blend_radius_m)
    movel([0.102129, -1.372121, -2.580460, -0.759809, 1.570796, 1.672925],accel_mss,speed_ms,0,blend_radius_m)
    movel([0.103079, -1.371569, -2.580841, -0.759978, 1.570796, 1.673875],accel_mss,speed_ms,0,blend_radius_m)
    movel([0.103407, -1.371411, -2.580951, -0.760027, 1.570796, 1.674203],accel_mss,speed_ms,0,blend_radius_m)
    movel([0.103782, -1.371467, -2.580912, -0.760010, 1.570796, 1.674579],accel_mss,speed_ms,0,blend_radius_m)
    movel([0.103972, -1.371802, -2.580680, -0.759907, 1.570796, 1.674769],accel_mss,speed_ms,0,blend_radius_m)
    movel([0.104047, -1.372591, -2.580134, -0.759665, 1.570796, 1.674843],accel_mss,speed_ms,0,blend_radius_m)
    movel([0.104025, -1.373418, -2.579560, -0.759411, 1.570796, 1.674822],accel_mss,speed_ms,0,blend_radius_m)
    movel([0.103868, -1.373951, -2.579189, -0.759249, 1.570796, 1.674664],accel_mss,speed_ms,0,blend_radius_m)
    movel([0.103307, -1.374492, -2.578813, -0.759084, 1.570796, 1.674104],accel_mss,speed_ms,0,blend_radius_m)
    movel([0.100371, -1.375894, -2.577835, -0.758659, 1.570796, 1.671167],accel_mss,speed_ms,0,blend_radius_m)
    movel([0.097202, -1.377295, -2.576856, -0.758238, 1.570796, 1.667998],accel_mss,speed_ms,0,blend_radius_m)
    movel([0.094275, -1.378433, -2.576058, -0.757898, 1.570796, 1.665072],accel_mss,speed_ms,0,blend_radius_m)
    movel([0.091963, -1.379186, -2.575529, -0.757674, 1.570796, 1.662759],accel_mss,speed_ms,0,blend_radius_m)
    movel([0.088651, -1.380120, -2.574872, -0.757397, 1.570796, 1.659447],accel_mss,speed_ms,0,blend_radius_m)
    movel([0.085300, -1.380994, -2.574256, -0.757139, 1.570796, 1.656096],accel_mss,speed_ms,0,blend_radius_m)
    movel([0.082794, -1.381553, -2.573861, -0.756974, 1.570796, 1.653590],accel_mss,speed_ms,0,blend_radius_m)
    movel([0.080908, -1.381888, -2.573625, -0.756876, 1.570796, 1.651704],accel_mss,speed_ms,0,blend_radius_m)
    movel([0.078698, -1.382220, -2.573390, -0.756779, 1.570796, 1.649495],accel_mss,speed_ms,0,blend_radius_m)
    movel([0.076615, -1.382497, -2.573195, -0.756698, 1.570796, 1.647412],accel_mss,speed_ms,0,blend_radius_m)
    movel([0.075933, -1.382504, -2.573189, -0.756696, 1.570796, 1.646730],accel_mss,speed_ms,0,blend_radius_m)
    movel([0.075687, -1.382338, -2.573307, -0.756744, 1.570796, 1.646483],accel_mss,speed_ms,0,blend_radius_m)
    movel([0.075673, -1.382108, -2.573469, -0.756812, 1.570796, 1.646469],accel_mss,speed_ms,0,blend_radius_m)
    movel([0.075722, -1.381504, -2.573896, -0.756989, 1.570796, 1.646518],accel_mss,speed_ms,0,blend_radius_m)
    movel([0.075826, -1.380764, -2.574419, -0.757207, 1.570796, 1.646623],accel_mss,speed_ms,0,blend_radius_m)
    movel([0.075986, -1.380177, -2.574832, -0.757380, 1.570796, 1.646783],accel_mss,speed_ms,0,blend_radius_m)
    movel([0.076193, -1.379748, -2.575134, -0.757507, 1.570796, 1.646990],accel_mss,speed_ms,0,blend_radius_m)
    movel([0.076445, -1.379509, -2.575302, -0.757578, 1.570796, 1.647241],accel_mss,speed_ms,0,blend_radius_m)
    movel([0.076934, -1.379415, -2.575368, -0.757606, 1.570796, 1.647730],accel_mss,speed_ms,0,blend_radius_m)
    movel([0.077336, -1.379386, -2.575388, -0.757614, 1.570796, 1.648132],accel_mss,speed_ms,0,blend_radius_m)
    movel([0.077768, -1.379376, -2.575395, -0.757617, 1.570796, 1.648564],accel_mss,speed_ms,0,blend_radius_m)
    movel([0.078966, -1.379343, -2.575419, -0.757627, 1.570796, 1.649762],accel_mss,speed_ms,0,blend_radius_m)
    movel([0.080402, -1.379226, -2.575501, -0.757662, 1.570796, 1.651198],accel_mss,speed_ms,0,blend_radius_m)
    movel([0.081934, -1.379044, -2.575629, -0.757716, 1.570796, 1.652730],accel_mss,speed_ms,0,blend_radius_m)
    movel([0.083427, -1.378810, -2.575794, -0.757786, 1.570796, 1.654223],accel_mss,speed_ms,0,blend_radius_m)
    movel([0.085813, -1.378280, -2.576166, -0.757944, 1.570796, 1.656609],accel_mss,speed_ms,0,blend_radius_m)
    movel([0.089434, -1.377259, -2.576881, -0.758249, 1.570796, 1.660230],accel_mss,speed_ms,0,blend_radius_m)
    movel([0.093095, -1.376133, -2.577668, -0.758587, 1.570796, 1.663891],accel_mss,speed_ms,0,blend_radius_m)
    speed_ms = 0.003
    movel([0.093095, -1.363017, -2.571624, -0.777747, 1.570796, 1.663891],accel_mss,speed_ms,0,blend_radius_m)
    speed_ms = 1.000
    movel([0.093095, -1.337880, -2.559143, -0.815367, 1.570796, 1.663891],accel_mss,speed_ms,0,blend_radius_m)
    movel([0.094637, -1.340831, -2.557189, -0.814369, 1.570796, 1.665433],accel_mss,speed_ms,0,blend_radius_m)
    movel([0.094637, -1.365917, -2.569633, -0.776839, 1.570796, 1.665433],accel_mss,speed_ms,0,blend_radius_m)
    speed_ms = 0.003
    movel([0.094637, -1.375697, -2.574164, -0.762527, 1.570796, 1.665433],accel_mss,speed_ms,0,blend_radius_m)
    speed_ms = 0.007
    movel([0.094653, -1.376219, -2.573799, -0.762371, 1.570796, 1.665449],accel_mss,speed_ms,0,blend_radius_m)
    movel([0.094666, -1.376607, -2.573528, -0.762254, 1.570796, 1.665463],accel_mss,speed_ms,0,blend_radius_m)
    movel([0.094670, -1.376842, -2.573363, -0.762184, 1.570796, 1.665466],accel_mss,speed_ms,0,blend_radius_m)
    movel([0.094469, -1.377074, -2.573201, -0.762115, 1.570796, 1.665265],accel_mss,speed_ms,0,blend_radius_m)
    movel([0.094064, -1.377312, -2.573034, -0.762044, 1.570796, 1.664860],accel_mss,speed_ms,0,blend_radius_m)
    movel([0.090980, -1.378254, -2.572372, -0.761763, 1.570796, 1.661777],accel_mss,speed_ms,0,blend_radius_m)
    movel([0.088110, -1.379102, -2.571776, -0.761511, 1.570796, 1.658906],accel_mss,speed_ms,0,blend_radius_m)
    movel([0.086332, -1.379547, -2.571462, -0.761379, 1.570796, 1.657129],accel_mss,speed_ms,0,blend_radius_m)
    movel([0.085492, -1.379705, -2.571351, -0.761333, 1.570796, 1.656288],accel_mss,speed_ms,0,blend_radius_m)
    movel([0.085165, -1.379666, -2.571378, -0.761344, 1.570796, 1.655961],accel_mss,speed_ms,0,blend_radius_m)
    movel([0.085064, -1.379455, -2.571527, -0.761407, 1.570796, 1.655861],accel_mss,speed_ms,0,blend_radius_m)
    movel([0.085171, -1.378948, -2.571884, -0.761557, 1.570796, 1.655967],accel_mss,speed_ms,0,blend_radius_m)
    movel([0.085340, -1.378391, -2.572276, -0.761722, 1.570796, 1.656137],accel_mss,speed_ms,0,blend_radius_m)
    movel([0.089986, -1.377037, -2.573226, -0.762125, 1.570796, 1.660782],accel_mss,speed_ms,0,blend_radius_m)
    movel([0.094637, -1.375697, -2.574164, -0.762527, 1.570796, 1.665433],accel_mss,speed_ms,0,blend_radius_m)
    speed_ms = 0.003
    movel([0.094637, -1.379003, -2.575658, -0.757728, 1.570796, 1.665433],accel_mss,speed_ms,0,blend_radius_m)
    speed_ms = 0.007
    movel([0.094653, -1.379524, -2.575292, -0.757573, 1.570796, 1.665449],accel_mss,speed_ms,0,blend_radius_m)
    movel([0.094666, -1.379910, -2.575020, -0.757459, 1.570796, 1.665463],accel_mss,speed_ms,0,blend_radius_m)
    movel([0.094670, -1.380144, -2.574855, -0.757390, 1.570796, 1.665466],accel_mss,speed_ms,0,blend_radius_m)
    movel([0.094469, -1.380376, -2.574692, -0.757321, 1.570796, 1.665265],accel_mss,speed_ms,0,blend_radius_m)
    movel([0.094064, -1.380613, -2.574525, -0.757251, 1.570796, 1.664860],accel_mss,speed_ms,0,blend_radius_m)
    movel([0.090980, -1.381553, -2.573862, -0.756974, 1.570796, 1.661777],accel_mss,speed_ms,0,blend_radius_m)
    movel([0.088110, -1.382398, -2.573264, -0.756727, 1.570796, 1.658906],accel_mss,speed_ms,0,blend_radius_m)
    movel([0.086332, -1.382843, -2.572950, -0.756597, 1.570796, 1.657129],accel_mss,speed_ms,0,blend_radius_m)
    movel([0.085492, -1.382999, -2.572838, -0.756551, 1.570796, 1.656288],accel_mss,speed_ms,0,blend_radius_m)
    movel([0.085165, -1.382961, -2.572866, -0.756562, 1.570796, 1.655961],accel_mss,speed_ms,0,blend_radius_m)
    movel([0.085064, -1.382750, -2.573015, -0.756624, 1.570796, 1.655861],accel_mss,speed_ms,0,blend_radius_m)
    movel([0.085171, -1.382245, -2.573372, -0.756771, 1.570796, 1.655967],accel_mss,speed_ms,0,blend_radius_m)
    movel([0.085340, -1.381689, -2.573765, -0.756934, 1.570796, 1.656137],accel_mss,speed_ms,0,blend_radius_m)
    movel([0.089986, -1.380339, -2.574718, -0.757332, 1.570796, 1.660782],accel_mss,speed_ms,0,blend_radius_m)
    movel([0.094637, -1.379003, -2.575658, -0.757728, 1.570796, 1.665433],accel_mss,speed_ms,0,blend_radius_m)
    speed_ms = 0.003
    movel([0.094637, -1.365917, -2.569633, -0.776839, 1.570796, 1.665433],accel_mss,speed_ms,0,blend_radius_m)
    speed_ms = 1.000
    movel([0.094637, -1.340831, -2.557189, -0.814369, 1.570796, 1.665433],accel_mss,speed_ms,0,blend_radius_m)
    movel([0.094776, -1.347374, -2.552816, -0.812199, 1.570796, 1.665572],accel_mss,speed_ms,0,blend_radius_m)
    movel([0.094776, -1.372344, -2.565176, -0.774868, 1.570796, 1.665572],accel_mss,speed_ms,0,blend_radius_m)
    speed_ms = 0.003
    movel([0.094776, -1.382075, -2.569677, -0.760637, 1.570796, 1.665572],accel_mss,speed_ms,0,blend_radius_m)
    speed_ms = 0.007
    movel([0.096440, -1.381462, -2.570110, -0.760816, 1.570796, 1.667237],accel_mss,speed_ms,0,blend_radius_m)
    movel([0.096911, -1.381238, -2.570269, -0.760882, 1.570796, 1.667707],accel_mss,speed_ms,0,blend_radius_m)
    movel([0.097314, -1.381204, -2.570293, -0.760892, 1.570796, 1.668110],accel_mss,speed_ms,0,blend_radius_m)
    movel([0.097422, -1.381359, -2.570183, -0.760846, 1.570796, 1.668218],accel_mss,speed_ms,0,blend_radius_m)
    movel([0.097435, -1.381607, -2.570008, -0.760774, 1.570796, 1.668231],accel_mss,speed_ms,0,blend_radius_m)
    movel([0.097301, -1.382148, -2.569625, -0.760616, 1.570796, 1.668098],accel_mss,speed_ms,0,blend_radius_m)
    movel([0.097178, -1.382558, -2.569334, -0.760496, 1.570796, 1.667974],accel_mss,speed_ms,0,blend_radius_m)
    movel([0.097039, -1.382977, -2.569037, -0.760375, 1.570796, 1.667835],accel_mss,speed_ms,0,blend_radius_m)
    movel([0.096697, -1.383916, -2.568371, -0.760103, 1.570796, 1.667493],accel_mss,speed_ms,0,blend_radius_m)
    movel([0.096287, -1.384945, -2.567638, -0.759806, 1.570796, 1.667084],accel_mss,speed_ms,0,blend_radius_m)
    movel([0.095880, -1.385915, -2.566946, -0.759527, 1.570796, 1.666677],accel_mss,speed_ms,0,blend_radius_m)
    movel([0.095733, -1.386137, -2.566788, -0.759464, 1.570796, 1.666529],accel_mss,speed_ms,0,blend_radius_m)
    movel([0.095575, -1.385999, -2.566887, -0.759503, 1.570796, 1.666371],accel_mss,speed_ms,0,blend_radius_m)
    movel([0.095465, -1.385691, -2.567106, -0.759592, 1.570796, 1.666261],accel_mss,speed_ms,0,blend_radius_m)
    movel([0.095361, -1.385540, -2.567214, -0.759635, 1.570796, 1.666157],accel_mss,speed_ms,0,blend_radius_m)
    movel([0.095087, -1.385336, -2.567360, -0.759694, 1.570796, 1.665884],accel_mss,speed_ms,0,blend_radius_m)
    movel([0.094829, -1.385186, -2.567466, -0.759737, 1.570796, 1.665625],accel_mss,speed_ms,0,blend_radius_m)
    movel([0.094690, -1.385009, -2.567592, -0.759787, 1.570796, 1.665486],accel_mss,speed_ms,0,blend_radius_m)
    movel([0.094486, -1.384711, -2.567805, -0.759873, 1.570796, 1.665282],accel_mss,speed_ms,0,blend_radius_m)
    movel([0.093913, -1.384330, -2.568076, -0.759983, 1.570796, 1.664709],accel_mss,speed_ms,0,blend_radius_m)
    movel([0.093257, -1.383995, -2.568314, -0.760080, 1.570796, 1.664053],accel_mss,speed_ms,0,blend_radius_m)
    movel([0.092692, -1.383834, -2.568428, -0.760126, 1.570796, 1.663488],accel_mss,speed_ms,0,blend_radius_m)
    movel([0.092049, -1.383769, -2.568475, -0.760145, 1.570796, 1.662845],accel_mss,speed_ms,0,blend_radius_m)
    movel([0.091353, -1.383774, -2.568471, -0.760144, 1.570796, 1.662149],accel_mss,speed_ms,0,blend_radius_m)
    movel([0.090674, -1.383839, -2.568425, -0.760125, 1.570796, 1.661470],accel_mss,speed_ms,0,blend_radius_m)
    movel([0.090083, -1.383966, -2.568335, -0.760088, 1.570796, 1.660879],accel_mss,speed_ms,0,blend_radius_m)
    movel([0.089683, -1.384047, -2.568277, -0.760065, 1.570796, 1.660479],accel_mss,speed_ms,0,blend_radius_m)
    movel([0.089967, -1.383735, -2.568499, -0.760155, 1.570796, 1.660763],accel_mss,speed_ms,0,blend_radius_m)
    movel([0.090498, -1.383539, -2.568638, -0.760212, 1.570796, 1.661294],accel_mss,speed_ms,0,blend_radius_m)
    movel([0.091427, -1.383232, -2.568856, -0.760301, 1.570796, 1.662224],accel_mss,speed_ms,0,blend_radius_m)
    movel([0.093010, -1.382702, -2.569233, -0.760455, 1.570796, 1.663806],accel_mss,speed_ms,0,blend_radius_m)
    movel([0.094776, -1.382075, -2.569677, -0.760637, 1.570796, 1.665572],accel_mss,speed_ms,0,blend_radius_m)
    speed_ms = 0.003
    movel([0.094776, -1.385364, -2.571160, -0.755866, 1.570796, 1.665572],accel_mss,speed_ms,0,blend_radius_m)
    speed_ms = 0.007
    movel([0.096440, -1.384753, -2.571594, -0.756042, 1.570796, 1.667237],accel_mss,speed_ms,0,blend_radius_m)
    movel([0.096911, -1.384529, -2.571754, -0.756107, 1.570796, 1.667707],accel_mss,speed_ms,0,blend_radius_m)
    movel([0.097314, -1.384495, -2.571778, -0.756117, 1.570796, 1.668110],accel_mss,speed_ms,0,blend_radius_m)
    movel([0.097422, -1.384650, -2.571667, -0.756072, 1.570796, 1.668218],accel_mss,speed_ms,0,blend_radius_m)
    movel([0.097435, -1.384896, -2.571492, -0.756001, 1.570796, 1.668231],accel_mss,speed_ms,0,blend_radius_m)
    movel([0.097301, -1.385436, -2.571108, -0.755845, 1.570796, 1.668098],accel_mss,speed_ms,0,blend_radius_m)
    movel([0.097178, -1.385846, -2.570816, -0.755727, 1.570796, 1.667974],accel_mss,speed_ms,0,blend_radius_m)
    movel([0.097039, -1.386263, -2.570519, -0.755607, 1.570796, 1.667835],accel_mss,speed_ms,0,blend_radius_m)
    movel([0.096697, -1.387199, -2.569851, -0.755339, 1.570796, 1.667493],accel_mss,speed_ms,0,blend_radius_m)
    movel([0.096287, -1.388225, -2.569117, -0.755047, 1.570796, 1.667084],accel_mss,speed_ms,0,blend_radius_m)
    movel([0.095880, -1.389193, -2.568423, -0.754773, 1.570796, 1.666677],accel_mss,speed_ms,0,blend_radius_m)
    movel([0.095733, -1.389415, -2.568264, -0.754710, 1.570796, 1.666529],accel_mss,speed_ms,0,blend_radius_m)
    movel([0.095575, -1.389277, -2.568363, -0.754749, 1.570796, 1.666371],accel_mss,speed_ms,0,blend_radius_m)
    movel([0.095465, -1.388970, -2.568583, -0.754836, 1.570796, 1.666261],accel_mss,speed_ms,0,blend_radius_m)
    movel([0.095361, -1.388818, -2.568692, -0.754879, 1.570796, 1.666157],accel_mss,speed_ms,0,blend_radius_m)
    movel([0.095087, -1.388615, -2.568837, -0.754936, 1.570796, 1.665884],accel_mss,speed_ms,0,blend_radius_m)
    movel([0.094829, -1.388466, -2.568945, -0.754979, 1.570796, 1.665625],accel_mss,speed_ms,0,blend_radius_m)
    movel([0.094690, -1.388289, -2.569071, -0.755029, 1.570796, 1.665486],accel_mss,speed_ms,0,blend_radius_m)
    movel([0.094486, -1.387992, -2.569284, -0.755113, 1.570796, 1.665282],accel_mss,speed_ms,0,blend_radius_m)
    movel([0.093913, -1.387612, -2.569556, -0.755221, 1.570796, 1.664709],accel_mss,speed_ms,0,blend_radius_m)
    movel([0.093257, -1.387278, -2.569794, -0.755317, 1.570796, 1.664053],accel_mss,speed_ms,0,blend_radius_m)
    movel([0.092692, -1.387118, -2.569909, -0.755362, 1.570796, 1.663488],accel_mss,speed_ms,0,blend_radius_m)
    movel([0.092049, -1.387053, -2.569955, -0.755381, 1.570796, 1.662845],accel_mss,speed_ms,0,blend_radius_m)
    movel([0.091353, -1.387058, -2.569952, -0.755379, 1.570796, 1.662149],accel_mss,speed_ms,0,blend_radius_m)
    movel([0.090674, -1.387122, -2.569906, -0.755361, 1.570796, 1.661470],accel_mss,speed_ms,0,blend_radius_m)
    movel([0.090083, -1.387249, -2.569815, -0.755325, 1.570796, 1.660879],accel_mss,speed_ms,0,blend_radius_m)
    movel([0.089683, -1.387330, -2.569757, -0.755302, 1.570796, 1.660479],accel_mss,speed_ms,0,blend_radius_m)
    movel([0.089967, -1.387019, -2.569980, -0.755391, 1.570796, 1.660763],accel_mss,speed_ms,0,blend_radius_m)
    movel([0.090498, -1.386824, -2.570119, -0.755446, 1.570796, 1.661294],accel_mss,speed_ms,0,blend_radius_m)
    movel([0.091427, -1.386517, -2.570338, -0.755534, 1.570796, 1.662224],accel_mss,speed_ms,0,blend_radius_m)
    movel([0.093010, -1.385988, -2.570715, -0.755686, 1.570796, 1.663806],accel_mss,speed_ms,0,blend_radius_m)
    movel([0.094776, -1.385364, -2.571160, -0.755866, 1.570796, 1.665572],accel_mss,speed_ms,0,blend_radius_m)
    speed_ms = 0.003
    movel([0.094776, -1.372344, -2.565176, -0.774868, 1.570796, 1.665572],accel_mss,speed_ms,0,blend_radius_m)
    speed_ms = 1.000
    movel([0.094776, -1.347374, -2.552816, -0.812199, 1.570796, 1.665572],accel_mss,speed_ms,0,blend_radius_m)
    movel([0.095070, -1.346731, -2.553248, -0.812409, 1.570796, 1.665866],accel_mss,speed_ms,0,blend_radius_m)
    movel([0.095070, -1.371713, -2.565617, -0.775059, 1.570796, 1.665866],accel_mss,speed_ms,0,blend_radius_m)
    speed_ms = 0.003
    movel([0.095070, -1.381449, -2.570120, -0.760820, 1.570796, 1.665866],accel_mss,speed_ms,0,blend_radius_m)
    speed_ms = 0.007
    movel([0.096152, -1.381011, -2.570430, -0.760949, 1.570796, 1.666948],accel_mss,speed_ms,0,blend_radius_m)
    movel([0.097416, -1.380470, -2.570812, -0.761108, 1.570796, 1.668212],accel_mss,speed_ms,0,blend_radius_m)
    movel([0.097749, -1.380346, -2.570899, -0.761144, 1.570796, 1.668546],accel_mss,speed_ms,0,blend_radius_m)
    movel([0.098110, -1.380392, -2.570867, -0.761131, 1.570796, 1.668906],accel_mss,speed_ms,0,blend_radius_m)
    movel([0.098230, -1.380590, -2.570727, -0.761072, 1.570796, 1.669026],accel_mss,speed_ms,0,blend_radius_m)
    movel([0.098219, -1.380960, -2.570466, -0.760964, 1.570796, 1.669016],accel_mss,speed_ms,0,blend_radius_m)
    movel([0.098079, -1.381576, -2.570030, -0.760783, 1.570796, 1.668875],accel_mss,speed_ms,0,blend_radius_m)
    movel([0.097743, -1.382661, -2.569262, -0.760467, 1.570796, 1.668540],accel_mss,speed_ms,0,blend_radius_m)
    movel([0.097071, -1.384490, -2.567962, -0.759937, 1.570796, 1.667867],accel_mss,speed_ms,0,blend_radius_m)
    movel([0.096148, -1.386582, -2.566470, -0.759337, 1.570796, 1.666944],accel_mss,speed_ms,0,blend_radius_m)
    movel([0.095198, -1.388510, -2.565090, -0.758790, 1.570796, 1.665994],accel_mss,speed_ms,0,blend_radius_m)
    movel([0.094651, -1.389228, -2.564574, -0.758587, 1.570796, 1.665447],accel_mss,speed_ms,0,blend_radius_m)
    movel([0.094291, -1.389485, -2.564389, -0.758515, 1.570796, 1.665088],accel_mss,speed_ms,0,blend_radius_m)
    movel([0.093555, -1.389857, -2.564122, -0.758410, 1.570796, 1.664352],accel_mss,speed_ms,0,blend_radius_m)
    movel([0.092679, -1.390248, -2.563840, -0.758301, 1.570796, 1.663475],accel_mss,speed_ms,0,blend_radius_m)
    movel([0.091771, -1.390598, -2.563588, -0.758203, 1.570796, 1.662567],accel_mss,speed_ms,0,blend_radius_m)
    movel([0.091344, -1.390760, -2.563472, -0.758158, 1.570796, 1.662140],accel_mss,speed_ms,0,blend_radius_m)
    movel([0.091077, -1.390880, -2.563385, -0.758124, 1.570796, 1.661873],accel_mss,speed_ms,0,blend_radius_m)
    movel([0.090865, -1.391070, -2.563248, -0.758071, 1.570796, 1.661661],accel_mss,speed_ms,0,blend_radius_m)
    movel([0.091295, -1.391060, -2.563255, -0.758074, 1.570796, 1.662091],accel_mss,speed_ms,0,blend_radius_m)
    movel([0.091815, -1.390883, -2.563383, -0.758123, 1.570796, 1.662611],accel_mss,speed_ms,0,blend_radius_m)
    movel([0.092251, -1.390721, -2.563500, -0.758169, 1.570796, 1.663048],accel_mss,speed_ms,0,blend_radius_m)
    movel([0.092769, -1.390519, -2.563645, -0.758225, 1.570796, 1.663566],accel_mss,speed_ms,0,blend_radius_m)
    movel([0.093283, -1.390311, -2.563795, -0.758283, 1.570796, 1.664079],accel_mss,speed_ms,0,blend_radius_m)
    movel([0.093711, -1.390127, -2.563927, -0.758335, 1.570796, 1.664507],accel_mss,speed_ms,0,blend_radius_m)
    movel([0.094299, -1.389872, -2.564111, -0.758406, 1.570796, 1.665096],accel_mss,speed_ms,0,blend_radius_m)
    movel([0.094706, -1.389789, -2.564171, -0.758429, 1.570796, 1.665503],accel_mss,speed_ms,0,blend_radius_m)
    movel([0.094972, -1.389962, -2.564046, -0.758381, 1.570796, 1.665769],accel_mss,speed_ms,0,blend_radius_m)
    movel([0.095076, -1.390324, -2.563786, -0.758280, 1.570796, 1.665873],accel_mss,speed_ms,0,blend_radius_m)
    movel([0.095081, -1.390609, -2.563580, -0.758200, 1.570796, 1.665877],accel_mss,speed_ms,0,blend_radius_m)
    movel([0.095059, -1.390956, -2.563330, -0.758103, 1.570796, 1.665855],accel_mss,speed_ms,0,blend_radius_m)
    movel([0.094920, -1.391327, -2.563063, -0.758000, 1.570796, 1.665716],accel_mss,speed_ms,0,blend_radius_m)
    movel([0.093941, -1.392067, -2.562528, -0.757794, 1.570796, 1.664738],accel_mss,speed_ms,0,blend_radius_m)
    movel([0.092368, -1.392707, -2.562066, -0.757617, 1.570796, 1.663164],accel_mss,speed_ms,0,blend_radius_m)
    movel([0.090193, -1.393424, -2.561546, -0.757419, 1.570796, 1.660989],accel_mss,speed_ms,0,blend_radius_m)
    movel([0.087277, -1.394246, -2.560950, -0.757193, 1.570796, 1.658074],accel_mss,speed_ms,0,blend_radius_m)
    movel([0.085160, -1.394791, -2.560554, -0.757044, 1.570796, 1.655956],accel_mss,speed_ms,0,blend_radius_m)
    movel([0.083595, -1.395139, -2.560301, -0.756949, 1.570796, 1.654391],accel_mss,speed_ms,0,blend_radius_m)
    movel([0.082460, -1.395328, -2.560164, -0.756897, 1.570796, 1.653257],accel_mss,speed_ms,0,blend_radius_m)
    movel([0.081822, -1.395320, -2.560169, -0.756899, 1.570796, 1.652619],accel_mss,speed_ms,0,blend_radius_m)
    movel([0.081641, -1.395219, -2.560243, -0.756927, 1.570796, 1.652437],accel_mss,speed_ms,0,blend_radius_m)
    movel([0.081532, -1.395035, -2.560377, -0.756977, 1.570796, 1.652328],accel_mss,speed_ms,0,blend_radius_m)
    movel([0.081519, -1.394687, -2.560630, -0.757072, 1.570796, 1.652316],accel_mss,speed_ms,0,blend_radius_m)
    movel([0.081608, -1.394239, -2.560955, -0.757195, 1.570796, 1.652404],accel_mss,speed_ms,0,blend_radius_m)
    movel([0.081764, -1.393806, -2.561269, -0.757314, 1.570796, 1.652560],accel_mss,speed_ms,0,blend_radius_m)
    movel([0.081959, -1.393518, -2.561478, -0.757393, 1.570796, 1.652756],accel_mss,speed_ms,0,blend_radius_m)
    movel([0.082312, -1.393264, -2.561662, -0.757463, 1.570796, 1.653108],accel_mss,speed_ms,0,blend_radius_m)
    movel([0.082560, -1.393207, -2.561703, -0.757479, 1.570796, 1.653356],accel_mss,speed_ms,0,blend_radius_m)
    movel([0.083142, -1.393136, -2.561755, -0.757498, 1.570796, 1.653938],accel_mss,speed_ms,0,blend_radius_m)
    movel([0.083870, -1.393046, -2.561820, -0.757523, 1.570796, 1.654666],accel_mss,speed_ms,0,blend_radius_m)
    movel([0.084273, -1.392965, -2.561878, -0.757545, 1.570796, 1.655069],accel_mss,speed_ms,0,blend_radius_m)
    movel([0.084581, -1.392758, -2.562029, -0.757603, 1.570796, 1.655377],accel_mss,speed_ms,0,blend_radius_m)
    movel([0.084311, -1.392695, -2.562074, -0.757620, 1.570796, 1.655108],accel_mss,speed_ms,0,blend_radius_m)
    movel([0.083989, -1.392708, -2.562065, -0.757616, 1.570796, 1.654785],accel_mss,speed_ms,0,blend_radius_m)
    movel([0.083558, -1.392751, -2.562033, -0.757604, 1.570796, 1.654354],accel_mss,speed_ms,0,blend_radius_m)
    movel([0.083144, -1.392794, -2.562002, -0.757593, 1.570796, 1.653940],accel_mss,speed_ms,0,blend_radius_m)
    movel([0.082748, -1.392818, -2.561985, -0.757586, 1.570796, 1.653545],accel_mss,speed_ms,0,blend_radius_m)
    movel([0.082417, -1.392823, -2.561981, -0.757585, 1.570796, 1.653213],accel_mss,speed_ms,0,blend_radius_m)
    movel([0.081839, -1.392468, -2.562239, -0.757683, 1.570796, 1.652636],accel_mss,speed_ms,0,blend_radius_m)
    movel([0.081234, -1.391081, -2.563240, -0.758068, 1.570796, 1.652030],accel_mss,speed_ms,0,blend_radius_m)
    movel([0.080689, -1.389524, -2.564361, -0.758504, 1.570796, 1.651485],accel_mss,speed_ms,0,blend_radius_m)
    movel([0.080352, -1.388078, -2.565399, -0.758912, 1.570796, 1.651148],accel_mss,speed_ms,0,blend_radius_m)
    movel([0.080191, -1.386915, -2.566232, -0.759242, 1.570796, 1.650987],accel_mss,speed_ms,0,blend_radius_m)
    movel([0.080184, -1.386139, -2.566786, -0.759463, 1.570796, 1.650980],accel_mss,speed_ms,0,blend_radius_m)
    movel([0.080307, -1.385620, -2.567157, -0.759612, 1.570796, 1.651104],accel_mss,speed_ms,0,blend_radius_m)
    movel([0.080582, -1.385323, -2.567369, -0.759697, 1.570796, 1.651378],accel_mss,speed_ms,0,blend_radius_m)
    movel([0.081195, -1.385168, -2.567479, -0.759742, 1.570796, 1.651991],accel_mss,speed_ms,0,blend_radius_m)
    movel([0.081739, -1.385071, -2.567548, -0.759770, 1.570796, 1.652535],accel_mss,speed_ms,0,blend_radius_m)
    movel([0.082338, -1.384981, -2.567612, -0.759795, 1.570796, 1.653134],accel_mss,speed_ms,0,blend_radius_m)
    movel([0.083396, -1.384803, -2.567739, -0.759847, 1.570796, 1.654192],accel_mss,speed_ms,0,blend_radius_m)
    movel([0.084436, -1.384567, -2.567907, -0.759915, 1.570796, 1.655232],accel_mss,speed_ms,0,blend_radius_m)
    movel([0.085955, -1.384156, -2.568200, -0.760033, 1.570796, 1.656751],accel_mss,speed_ms,0,blend_radius_m)
    movel([0.089220, -1.383220, -2.568865, -0.760304, 1.570796, 1.660017],accel_mss,speed_ms,0,blend_radius_m)
    movel([0.092482, -1.382280, -2.569531, -0.760578, 1.570796, 1.663278],accel_mss,speed_ms,0,blend_radius_m)
    movel([0.094013, -1.381815, -2.569861, -0.760713, 1.570796, 1.664810],accel_mss,speed_ms,0,blend_radius_m)
    movel([0.095070, -1.381449, -2.570120, -0.760820, 1.570796, 1.665866],accel_mss,speed_ms,0,blend_radius_m)
    speed_ms = 0.003
    movel([0.095070, -1.384739, -2.571604, -0.756046, 1.570796, 1.665866],accel_mss,speed_ms,0,blend_radius_m)
    speed_ms = 0.007
    movel([0.096152, -1.384302, -2.571915, -0.756172, 1.570796, 1.666948],accel_mss,speed_ms,0,blend_radius_m)
    movel([0.097416, -1.383762, -2.572298, -0.756329, 1.570796, 1.668212],accel_mss,speed_ms,0,blend_radius_m)
    movel([0.097749, -1.383640, -2.572385, -0.756365, 1.570796, 1.668546],accel_mss,speed_ms,0,blend_radius_m)
    movel([0.098110, -1.383685, -2.572353, -0.756352, 1.570796, 1.668906],accel_mss,speed_ms,0,blend_radius_m)
    movel([0.098230, -1.383883, -2.572212, -0.756294, 1.570796, 1.669026],accel_mss,speed_ms,0,blend_radius_m)
    movel([0.098219, -1.384251, -2.571951, -0.756187, 1.570796, 1.669016],accel_mss,speed_ms,0,blend_radius_m)
    movel([0.098079, -1.384866, -2.571514, -0.756009, 1.570796, 1.668875],accel_mss,speed_ms,0,blend_radius_m)
    movel([0.097743, -1.385947, -2.570744, -0.755698, 1.570796, 1.668540],accel_mss,speed_ms,0,blend_radius_m)
    movel([0.097071, -1.387772, -2.569442, -0.755176, 1.570796, 1.667867],accel_mss,speed_ms,0,blend_radius_m)
    movel([0.096148, -1.389858, -2.567946, -0.754585, 1.570796, 1.666944],accel_mss,speed_ms,0,blend_radius_m)
    movel([0.095198, -1.391781, -2.566562, -0.754046, 1.570796, 1.665994],accel_mss,speed_ms,0,blend_radius_m)
    movel([0.094651, -1.392496, -2.566046, -0.753847, 1.570796, 1.665447],accel_mss,speed_ms,0,blend_radius_m)
    movel([0.094291, -1.392753, -2.565860, -0.753775, 1.570796, 1.665088],accel_mss,speed_ms,0,blend_radius_m)
    movel([0.093555, -1.393124, -2.565592, -0.753673, 1.570796, 1.664352],accel_mss,speed_ms,0,blend_radius_m)
    movel([0.092679, -1.393514, -2.565310, -0.753565, 1.570796, 1.663475],accel_mss,speed_ms,0,blend_radius_m)
    movel([0.091771, -1.393863, -2.565057, -0.753469, 1.570796, 1.662567],accel_mss,speed_ms,0,blend_radius_m)
    movel([0.091344, -1.394024, -2.564941, -0.753424, 1.570796, 1.662140],accel_mss,speed_ms,0,blend_radius_m)
    movel([0.091077, -1.394144, -2.564854, -0.753391, 1.570796, 1.661873],accel_mss,speed_ms,0,blend_radius_m)
    movel([0.090865, -1.394334, -2.564717, -0.753339, 1.570796, 1.661661],accel_mss,speed_ms,0,blend_radius_m)
    movel([0.091295, -1.394324, -2.564724, -0.753342, 1.570796, 1.662091],accel_mss,speed_ms,0,blend_radius_m)
    movel([0.091815, -1.394147, -2.564852, -0.753390, 1.570796, 1.662611],accel_mss,speed_ms,0,blend_radius_m)
    movel([0.092251, -1.393985, -2.564969, -0.753435, 1.570796, 1.663048],accel_mss,speed_ms,0,blend_radius_m)
    movel([0.092769, -1.393785, -2.565114, -0.753490, 1.570796, 1.663566],accel_mss,speed_ms,0,blend_radius_m)
    movel([0.093283, -1.393577, -2.565264, -0.753547, 1.570796, 1.664079],accel_mss,speed_ms,0,blend_radius_m)
    movel([0.093711, -1.393394, -2.565397, -0.753598, 1.570796, 1.664507],accel_mss,speed_ms,0,blend_radius_m)
    movel([0.094299, -1.393139, -2.565582, -0.753669, 1.570796, 1.665096],accel_mss,speed_ms,0,blend_radius_m)
    movel([0.094706, -1.393056, -2.565641, -0.753692, 1.570796, 1.665503],accel_mss,speed_ms,0,blend_radius_m)
    movel([0.094972, -1.393229, -2.565516, -0.753644, 1.570796, 1.665769],accel_mss,speed_ms,0,blend_radius_m)
    movel([0.095076, -1.393589, -2.565255, -0.753544, 1.570796, 1.665873],accel_mss,speed_ms,0,blend_radius_m)
    movel([0.095081, -1.393874, -2.565049, -0.753465, 1.570796, 1.665877],accel_mss,speed_ms,0,blend_radius_m)
    movel([0.095059, -1.394220, -2.564799, -0.753370, 1.570796, 1.665855],accel_mss,speed_ms,0,blend_radius_m)
    movel([0.094920, -1.394590, -2.564531, -0.753268, 1.570796, 1.665716],accel_mss,speed_ms,0,blend_radius_m)
    movel([0.093941, -1.395328, -2.563995, -0.753066, 1.570796, 1.664738],accel_mss,speed_ms,0,blend_radius_m)
    movel([0.092368, -1.395966, -2.563531, -0.752892, 1.570796, 1.663164],accel_mss,speed_ms,0,blend_radius_m)
    movel([0.090193, -1.396682, -2.563010, -0.752697, 1.570796, 1.660989],accel_mss,speed_ms,0,blend_radius_m)
    movel([0.087277, -1.397501, -2.562413, -0.752475, 1.570796, 1.658074],accel_mss,speed_ms,0,blend_radius_m)
    movel([0.085160, -1.398044, -2.562017, -0.752328, 1.570796, 1.655956],accel_mss,speed_ms,0,blend_radius_m)
    movel([0.083595, -1.398392, -2.561763, -0.752234, 1.570796, 1.654391],accel_mss,speed_ms,0,blend_radius_m)
    movel([0.082460, -1.398579, -2.561626, -0.752184, 1.570796, 1.653257],accel_mss,speed_ms,0,blend_radius_m)
    movel([0.081822, -1.398572, -2.561631, -0.752186, 1.570796, 1.652619],accel_mss,speed_ms,0,blend_radius_m)
    movel([0.081641, -1.398471, -2.561705, -0.752213, 1.570796, 1.652437],accel_mss,speed_ms,0,blend_radius_m)
    movel([0.081532, -1.398288, -2.561839, -0.752262, 1.570796, 1.652328],accel_mss,speed_ms,0,blend_radius_m)
    movel([0.081519, -1.397940, -2.562093, -0.752356, 1.570796, 1.652316],accel_mss,speed_ms,0,blend_radius_m)
    movel([0.081608, -1.397494, -2.562419, -0.752477, 1.570796, 1.652404],accel_mss,speed_ms,0,blend_radius_m)
    movel([0.081764, -1.397062, -2.562733, -0.752594, 1.570796, 1.652560],accel_mss,speed_ms,0,blend_radius_m)
    movel([0.081959, -1.396775, -2.562943, -0.752672, 1.570796, 1.652756],accel_mss,speed_ms,0,blend_radius_m)
    movel([0.082312, -1.396522, -2.563127, -0.752740, 1.570796, 1.653108],accel_mss,speed_ms,0,blend_radius_m)
    movel([0.082560, -1.396465, -2.563168, -0.752756, 1.570796, 1.653356],accel_mss,speed_ms,0,blend_radius_m)
    movel([0.083142, -1.396394, -2.563220, -0.752775, 1.570796, 1.653938],accel_mss,speed_ms,0,blend_radius_m)
    movel([0.083870, -1.396304, -2.563285, -0.752799, 1.570796, 1.654666],accel_mss,speed_ms,0,blend_radius_m)
    movel([0.084273, -1.396224, -2.563344, -0.752821, 1.570796, 1.655069],accel_mss,speed_ms,0,blend_radius_m)
    movel([0.084581, -1.396017, -2.563494, -0.752878, 1.570796, 1.655377],accel_mss,speed_ms,0,blend_radius_m)
    movel([0.084311, -1.395955, -2.563540, -0.752895, 1.570796, 1.655108],accel_mss,speed_ms,0,blend_radius_m)
    movel([0.083989, -1.395967, -2.563531, -0.752891, 1.570796, 1.654785],accel_mss,speed_ms,0,blend_radius_m)
    movel([0.083558, -1.396010, -2.563499, -0.752880, 1.570796, 1.654354],accel_mss,speed_ms,0,blend_radius_m)
    movel([0.083144, -1.396053, -2.563468, -0.752868, 1.570796, 1.653940],accel_mss,speed_ms,0,blend_radius_m)
    movel([0.082748, -1.396077, -2.563451, -0.752862, 1.570796, 1.653545],accel_mss,speed_ms,0,blend_radius_m)
    movel([0.082417, -1.396082, -2.563447, -0.752860, 1.570796, 1.653213],accel_mss,speed_ms,0,blend_radius_m)
    movel([0.081839, -1.395727, -2.563705, -0.752957, 1.570796, 1.652636],accel_mss,speed_ms,0,blend_radius_m)
    movel([0.081234, -1.394344, -2.564709, -0.753336, 1.570796, 1.652030],accel_mss,speed_ms,0,blend_radius_m)
    movel([0.080689, -1.392792, -2.565832, -0.753765, 1.570796, 1.651485],accel_mss,speed_ms,0,blend_radius_m)
    movel([0.080352, -1.391350, -2.566872, -0.754166, 1.570796, 1.651148],accel_mss,speed_ms,0,blend_radius_m)
    movel([0.080191, -1.390190, -2.567708, -0.754492, 1.570796, 1.650987],accel_mss,speed_ms,0,blend_radius_m)
    movel([0.080184, -1.389417, -2.568263, -0.754709, 1.570796, 1.650980],accel_mss,speed_ms,0,blend_radius_m)
    movel([0.080307, -1.388898, -2.568635, -0.754856, 1.570796, 1.651104],accel_mss,speed_ms,0,blend_radius_m)
    movel([0.080582, -1.388603, -2.568847, -0.754940, 1.570796, 1.651378],accel_mss,speed_ms,0,blend_radius_m)
    movel([0.081195, -1.388448, -2.568957, -0.754984, 1.570796, 1.651991],accel_mss,speed_ms,0,blend_radius_m)
    movel([0.081739, -1.388352, -2.569026, -0.755011, 1.570796, 1.652535],accel_mss,speed_ms,0,blend_radius_m)
    movel([0.082338, -1.388262, -2.569091, -0.755036, 1.570796, 1.653134],accel_mss,speed_ms,0,blend_radius_m)
    movel([0.083396, -1.388084, -2.569218, -0.755087, 1.570796, 1.654192],accel_mss,speed_ms,0,blend_radius_m)
    movel([0.084436, -1.387849, -2.569386, -0.755154, 1.570796, 1.655232],accel_mss,speed_ms,0,blend_radius_m)
    movel([0.085955, -1.387438, -2.569680, -0.755271, 1.570796, 1.656751],accel_mss,speed_ms,0,blend_radius_m)
    movel([0.089220, -1.386505, -2.570346, -0.755538, 1.570796, 1.660017],accel_mss,speed_ms,0,blend_radius_m)
    movel([0.092482, -1.385568, -2.571014, -0.755807, 1.570796, 1.663278],accel_mss,speed_ms,0,blend_radius_m)
    movel([0.094013, -1.385104, -2.571344, -0.755940, 1.570796, 1.664810],accel_mss,speed_ms,0,blend_radius_m)
    movel([0.095070, -1.384739, -2.571604, -0.756046, 1.570796, 1.665866],accel_mss,speed_ms,0,blend_radius_m)
    speed_ms = 0.003
    movel([0.095070, -1.371713, -2.565617, -0.775059, 1.570796, 1.665866],accel_mss,speed_ms,0,blend_radius_m)
    speed_ms = 1.000
    movel([0.095070, -1.346731, -2.553248, -0.812409, 1.570796, 1.665866],accel_mss,speed_ms,0,blend_radius_m)
    movel([0.089293, -1.355826, -2.547083, -0.809480, 1.570796, 1.660089],accel_mss,speed_ms,0,blend_radius_m)
    movel([0.089293, -1.380644, -2.559336, -0.772409, 1.570796, 1.660089],accel_mss,speed_ms,0,blend_radius_m)
    speed_ms = 0.003
    movel([0.089293, -1.390310, -2.563795, -0.758283, 1.570796, 1.660089],accel_mss,speed_ms,0,blend_radius_m)
    speed_ms = 0.007
    movel([0.089533, -1.390446, -2.563697, -0.758245, 1.570796, 1.660329],accel_mss,speed_ms,0,blend_radius_m)
    movel([0.089491, -1.390735, -2.563490, -0.758165, 1.570796, 1.660287],accel_mss,speed_ms,0,blend_radius_m)
    movel([0.089053, -1.390950, -2.563335, -0.758105, 1.570796, 1.659850],accel_mss,speed_ms,0,blend_radius_m)
    movel([0.088549, -1.391115, -2.563215, -0.758058, 1.570796, 1.659346],accel_mss,speed_ms,0,blend_radius_m)
    movel([0.088022, -1.391275, -2.563100, -0.758014, 1.570796, 1.658818],accel_mss,speed_ms,0,blend_radius_m)
    movel([0.087755, -1.391333, -2.563058, -0.757998, 1.570796, 1.658551],accel_mss,speed_ms,0,blend_radius_m)
    movel([0.087527, -1.391260, -2.563111, -0.758018, 1.570796, 1.658324],accel_mss,speed_ms,0,blend_radius_m)
    movel([0.087836, -1.390747, -2.563481, -0.758161, 1.570796, 1.658633],accel_mss,speed_ms,0,blend_radius_m)
    movel([0.088216, -1.390466, -2.563683, -0.758240, 1.570796, 1.659012],accel_mss,speed_ms,0,blend_radius_m)
    movel([0.088598, -1.390297, -2.563805, -0.758287, 1.570796, 1.659394],accel_mss,speed_ms,0,blend_radius_m)
    movel([0.088951, -1.390251, -2.563838, -0.758300, 1.570796, 1.659747],accel_mss,speed_ms,0,blend_radius_m)
    movel([0.089293, -1.390310, -2.563795, -0.758283, 1.570796, 1.660089],accel_mss,speed_ms,0,blend_radius_m)
    speed_ms = 0.003
    movel([0.089293, -1.393576, -2.565265, -0.753548, 1.570796, 1.660089],accel_mss,speed_ms,0,blend_radius_m)
    speed_ms = 0.007
    movel([0.089533, -1.393712, -2.565167, -0.753510, 1.570796, 1.660329],accel_mss,speed_ms,0,blend_radius_m)
    movel([0.089491, -1.393999, -2.564959, -0.753431, 1.570796, 1.660287],accel_mss,speed_ms,0,blend_radius_m)
    movel([0.089053, -1.394214, -2.564804, -0.753372, 1.570796, 1.659850],accel_mss,speed_ms,0,blend_radius_m)
    movel([0.088549, -1.394379, -2.564684, -0.753326, 1.570796, 1.659346],accel_mss,speed_ms,0,blend_radius_m)
    movel([0.088022, -1.394539, -2.564568, -0.753283, 1.570796, 1.658818],accel_mss,speed_ms,0,blend_radius_m)
    movel([0.087755, -1.394596, -2.564526, -0.753267, 1.570796, 1.658551],accel_mss,speed_ms,0,blend_radius_m)
    movel([0.087527, -1.394523, -2.564579, -0.753287, 1.570796, 1.658324],accel_mss,speed_ms,0,blend_radius_m)
    movel([0.087836, -1.394012, -2.564950, -0.753428, 1.570796, 1.658633],accel_mss,speed_ms,0,blend_radius_m)
    movel([0.088216, -1.393731, -2.565153, -0.753505, 1.570796, 1.659012],accel_mss,speed_ms,0,blend_radius_m)
    movel([0.088598, -1.393563, -2.565275, -0.753551, 1.570796, 1.659394],accel_mss,speed_ms,0,blend_radius_m)
    movel([0.088951, -1.393516, -2.565308, -0.753564, 1.570796, 1.659747],accel_mss,speed_ms,0,blend_radius_m)
    movel([0.089293, -1.393576, -2.565265, -0.753548, 1.570796, 1.660089],accel_mss,speed_ms,0,blend_radius_m)
    speed_ms = 0.003
    movel([0.089293, -1.380644, -2.559336, -0.772409, 1.570796, 1.660089],accel_mss,speed_ms,0,blend_radius_m)
    speed_ms = 1.000
    movel([0.089293, -1.355826, -2.547083, -0.809480, 1.570796, 1.660089],accel_mss,speed_ms,0,blend_radius_m)
    movel([0.088410, -1.349799, -2.551181, -0.811409, 1.570796, 1.659206],accel_mss,speed_ms,0,blend_radius_m)
    movel([0.088410, -1.374726, -2.563511, -0.774153, 1.570796, 1.659206],accel_mss,speed_ms,0,blend_radius_m)
    speed_ms = 0.003
    movel([0.088410, -1.384438, -2.567999, -0.759952, 1.570796, 1.659206],accel_mss,speed_ms,0,blend_radius_m)
    speed_ms = 0.007
    movel([0.087081, -1.384926, -2.567651, -0.759811, 1.570796, 1.657878],accel_mss,speed_ms,0,blend_radius_m)
    movel([0.085949, -1.385546, -2.567210, -0.759633, 1.570796, 1.656745],accel_mss,speed_ms,0,blend_radius_m)
    movel([0.084872, -1.386318, -2.566658, -0.759412, 1.570796, 1.655668],accel_mss,speed_ms,0,blend_radius_m)
    movel([0.083929, -1.387193, -2.566033, -0.759163, 1.570796, 1.654725],accel_mss,speed_ms,0,blend_radius_m)
    movel([0.083360, -1.387850, -2.565563, -0.758976, 1.570796, 1.654157],accel_mss,speed_ms,0,blend_radius_m)
    movel([0.082732, -1.388688, -2.564962, -0.758739, 1.570796, 1.653528],accel_mss,speed_ms,0,blend_radius_m)
    movel([0.082181, -1.389503, -2.564376, -0.758510, 1.570796, 1.652978],accel_mss,speed_ms,0,blend_radius_m)
    movel([0.081904, -1.390039, -2.563990, -0.758359, 1.570796, 1.652700],accel_mss,speed_ms,0,blend_radius_m)
    movel([0.081705, -1.390252, -2.563838, -0.758300, 1.570796, 1.652502],accel_mss,speed_ms,0,blend_radius_m)
    movel([0.081566, -1.390049, -2.563984, -0.758357, 1.570796, 1.652362],accel_mss,speed_ms,0,blend_radius_m)
    movel([0.081299, -1.389034, -2.564713, -0.758642, 1.570796, 1.652095],accel_mss,speed_ms,0,blend_radius_m)
    movel([0.081058, -1.387988, -2.565464, -0.758937, 1.570796, 1.651854],accel_mss,speed_ms,0,blend_radius_m)
    movel([0.080915, -1.387123, -2.566083, -0.759183, 1.570796, 1.651712],accel_mss,speed_ms,0,blend_radius_m)
    movel([0.080836, -1.386274, -2.566690, -0.759425, 1.570796, 1.651632],accel_mss,speed_ms,0,blend_radius_m)
    movel([0.080928, -1.385938, -2.566930, -0.759521, 1.570796, 1.651725],accel_mss,speed_ms,0,blend_radius_m)
    movel([0.081186, -1.385742, -2.567070, -0.759577, 1.570796, 1.651983],accel_mss,speed_ms,0,blend_radius_m)
    movel([0.081800, -1.385622, -2.567155, -0.759611, 1.570796, 1.652596],accel_mss,speed_ms,0,blend_radius_m)
    movel([0.082664, -1.385488, -2.567251, -0.759650, 1.570796, 1.653461],accel_mss,speed_ms,0,blend_radius_m)
    movel([0.083900, -1.385238, -2.567429, -0.759721, 1.570796, 1.654697],accel_mss,speed_ms,0,blend_radius_m)
    movel([0.085342, -1.384916, -2.567659, -0.759814, 1.570796, 1.656138],accel_mss,speed_ms,0,blend_radius_m)
    movel([0.086879, -1.384542, -2.567925, -0.759922, 1.570796, 1.657675],accel_mss,speed_ms,0,blend_radius_m)
    movel([0.087796, -1.384317, -2.568085, -0.759987, 1.570796, 1.658593],accel_mss,speed_ms,0,blend_radius_m)
    movel([0.088317, -1.384208, -2.568162, -0.760018, 1.570796, 1.659114],accel_mss,speed_ms,0,blend_radius_m)
    movel([0.088631, -1.384168, -2.568191, -0.760030, 1.570796, 1.659427],accel_mss,speed_ms,0,blend_radius_m)
    movel([0.088410, -1.384438, -2.567999, -0.759952, 1.570796, 1.659206],accel_mss,speed_ms,0,blend_radius_m)
    speed_ms = 0.003
    movel([0.088410, -1.387720, -2.569479, -0.755191, 1.570796, 1.659206],accel_mss,speed_ms,0,blend_radius_m)
    speed_ms = 0.007
    movel([0.087081, -1.388207, -2.569130, -0.755052, 1.570796, 1.657878],accel_mss,speed_ms,0,blend_radius_m)
    movel([0.085949, -1.388825, -2.568687, -0.754877, 1.570796, 1.656745],accel_mss,speed_ms,0,blend_radius_m)
    movel([0.084872, -1.389595, -2.568135, -0.754659, 1.570796, 1.655668],accel_mss,speed_ms,0,blend_radius_m)
    movel([0.083929, -1.390467, -2.567508, -0.754414, 1.570796, 1.654725],accel_mss,speed_ms,0,blend_radius_m)
    movel([0.083360, -1.391123, -2.567036, -0.754230, 1.570796, 1.654157],accel_mss,speed_ms,0,blend_radius_m)
    movel([0.082732, -1.391958, -2.566434, -0.753997, 1.570796, 1.653528],accel_mss,speed_ms,0,blend_radius_m)
    movel([0.082181, -1.392771, -2.565848, -0.753771, 1.570796, 1.652978],accel_mss,speed_ms,0,blend_radius_m)
    movel([0.081904, -1.393306, -2.565461, -0.753622, 1.570796, 1.652700],accel_mss,speed_ms,0,blend_radius_m)
    movel([0.081705, -1.393518, -2.565308, -0.753564, 1.570796, 1.652502],accel_mss,speed_ms,0,blend_radius_m)
    movel([0.081566, -1.393315, -2.565454, -0.753620, 1.570796, 1.652362],accel_mss,speed_ms,0,blend_radius_m)
    movel([0.081299, -1.392304, -2.566185, -0.753900, 1.570796, 1.652095],accel_mss,speed_ms,0,blend_radius_m)
    movel([0.081058, -1.391260, -2.566937, -0.754191, 1.570796, 1.651854],accel_mss,speed_ms,0,blend_radius_m)
    movel([0.080915, -1.390398, -2.567558, -0.754433, 1.570796, 1.651712],accel_mss,speed_ms,0,blend_radius_m)
    movel([0.080836, -1.389551, -2.568167, -0.754672, 1.570796, 1.651632],accel_mss,speed_ms,0,blend_radius_m)
    movel([0.080928, -1.389216, -2.568407, -0.754766, 1.570796, 1.651725],accel_mss,speed_ms,0,blend_radius_m)
    movel([0.081186, -1.389020, -2.568547, -0.754822, 1.570796, 1.651983],accel_mss,speed_ms,0,blend_radius_m)
    movel([0.081800, -1.388901, -2.568633, -0.754855, 1.570796, 1.652596],accel_mss,speed_ms,0,blend_radius_m)
    movel([0.082664, -1.388767, -2.568728, -0.754893, 1.570796, 1.653461],accel_mss,speed_ms,0,blend_radius_m)
    movel([0.083900, -1.388518, -2.568907, -0.754964, 1.570796, 1.654697],accel_mss,speed_ms,0,blend_radius_m)
    movel([0.085342, -1.388196, -2.569138, -0.755055, 1.570796, 1.656138],accel_mss,speed_ms,0,blend_radius_m)
    movel([0.086879, -1.387824, -2.569404, -0.755161, 1.570796, 1.657675],accel_mss,speed_ms,0,blend_radius_m)
    movel([0.087796, -1.387599, -2.569565, -0.755225, 1.570796, 1.658593],accel_mss,speed_ms,0,blend_radius_m)
    movel([0.088317, -1.387491, -2.569642, -0.755256, 1.570796, 1.659114],accel_mss,speed_ms,0,blend_radius_m)
    movel([0.088631, -1.387451, -2.569671, -0.755267, 1.570796, 1.659427],accel_mss,speed_ms,0,blend_radius_m)
    movel([0.088410, -1.387720, -2.569479, -0.755191, 1.570796, 1.659206],accel_mss,speed_ms,0,blend_radius_m)
    speed_ms = 0.003
    movel([0.088410, -1.374726, -2.563511, -0.774153, 1.570796, 1.659206],accel_mss,speed_ms,0,blend_radius_m)
    speed_ms = 1.000
    movel([0.088410, -1.349799, -2.551181, -0.811409, 1.570796, 1.659206],accel_mss,speed_ms,0,blend_radius_m)
    movel([0.072038, -1.358116, -2.545513, -0.808760, 1.570796, 1.642834],accel_mss,speed_ms,0,blend_radius_m)
    movel([0.072038, -1.382893, -2.557737, -0.771760, 1.570796, 1.642834],accel_mss,speed_ms,0,blend_radius_m)
    speed_ms = 0.003
    movel([0.072038, -1.392541, -2.562186, -0.757663, 1.570796, 1.642834],accel_mss,speed_ms,0,blend_radius_m)
    speed_ms = 0.007
    movel([0.072079, -1.392738, -2.562043, -0.757608, 1.570796, 1.642875],accel_mss,speed_ms,0,blend_radius_m)
    movel([0.071854, -1.393010, -2.561846, -0.757533, 1.570796, 1.642650],accel_mss,speed_ms,0,blend_radius_m)
    movel([0.071545, -1.393082, -2.561794, -0.757513, 1.570796, 1.642341],accel_mss,speed_ms,0,blend_radius_m)
    movel([0.071303, -1.393090, -2.561788, -0.757511, 1.570796, 1.642100],accel_mss,speed_ms,0,blend_radius_m)
    movel([0.071035, -1.393108, -2.561775, -0.757506, 1.570796, 1.641831],accel_mss,speed_ms,0,blend_radius_m)
    movel([0.070605, -1.393174, -2.561727, -0.757488, 1.570796, 1.641402],accel_mss,speed_ms,0,blend_radius_m)
    movel([0.070116, -1.393271, -2.561657, -0.757461, 1.570796, 1.640912],accel_mss,speed_ms,0,blend_radius_m)
    movel([0.069632, -1.393385, -2.561575, -0.757430, 1.570796, 1.640429],accel_mss,speed_ms,0,blend_radius_m)
    movel([0.068674, -1.393599, -2.561419, -0.757371, 1.570796, 1.639470],accel_mss,speed_ms,0,blend_radius_m)
    movel([0.068254, -1.393580, -2.561433, -0.757376, 1.570796, 1.639050],accel_mss,speed_ms,0,blend_radius_m)
    movel([0.068198, -1.393373, -2.561583, -0.757433, 1.570796, 1.638995],accel_mss,speed_ms,0,blend_radius_m)
    movel([0.068476, -1.392973, -2.561872, -0.757543, 1.570796, 1.639272],accel_mss,speed_ms,0,blend_radius_m)
    movel([0.068846, -1.392690, -2.562077, -0.757621, 1.570796, 1.639642],accel_mss,speed_ms,0,blend_radius_m)
    movel([0.069096, -1.392605, -2.562139, -0.757645, 1.570796, 1.639893],accel_mss,speed_ms,0,blend_radius_m)
    movel([0.069570, -1.392494, -2.562220, -0.757676, 1.570796, 1.640367],accel_mss,speed_ms,0,blend_radius_m)
    movel([0.070403, -1.392329, -2.562339, -0.757721, 1.570796, 1.641200],accel_mss,speed_ms,0,blend_radius_m)
    movel([0.071125, -1.392221, -2.562417, -0.757751, 1.570796, 1.641922],accel_mss,speed_ms,0,blend_radius_m)
    movel([0.071701, -1.392164, -2.562458, -0.757767, 1.570796, 1.642497],accel_mss,speed_ms,0,blend_radius_m)
    movel([0.071942, -1.392284, -2.562371, -0.757734, 1.570796, 1.642738],accel_mss,speed_ms,0,blend_radius_m)
    movel([0.072038, -1.392541, -2.562186, -0.757663, 1.570796, 1.642834],accel_mss,speed_ms,0,blend_radius_m)
    speed_ms = 0.003
    movel([0.072038, -1.395800, -2.563652, -0.752937, 1.570796, 1.642834],accel_mss,speed_ms,0,blend_radius_m)
    speed_ms = 0.007
    movel([0.072079, -1.395997, -2.563509, -0.752883, 1.570796, 1.642875],accel_mss,speed_ms,0,blend_radius_m)
    movel([0.071854, -1.396269, -2.563311, -0.752809, 1.570796, 1.642650],accel_mss,speed_ms,0,blend_radius_m)
    movel([0.071545, -1.396340, -2.563259, -0.752790, 1.570796, 1.642341],accel_mss,speed_ms,0,blend_radius_m)
    movel([0.071303, -1.396348, -2.563254, -0.752788, 1.570796, 1.642100],accel_mss,speed_ms,0,blend_radius_m)
    movel([0.071035, -1.396366, -2.563240, -0.752783, 1.570796, 1.641831],accel_mss,speed_ms,0,blend_radius_m)
    movel([0.070605, -1.396432, -2.563192, -0.752765, 1.570796, 1.641402],accel_mss,speed_ms,0,blend_radius_m)
    movel([0.070116, -1.396529, -2.563122, -0.752738, 1.570796, 1.640912],accel_mss,speed_ms,0,blend_radius_m)
    movel([0.069632, -1.396642, -2.563039, -0.752708, 1.570796, 1.640429],accel_mss,speed_ms,0,blend_radius_m)
    movel([0.068674, -1.396856, -2.562883, -0.752649, 1.570796, 1.639470],accel_mss,speed_ms,0,blend_radius_m)
    movel([0.068254, -1.396836, -2.562898, -0.752655, 1.570796, 1.639050],accel_mss,speed_ms,0,blend_radius_m)
    movel([0.068198, -1.396630, -2.563048, -0.752711, 1.570796, 1.638995],accel_mss,speed_ms,0,blend_radius_m)
    movel([0.068476, -1.396232, -2.563338, -0.752819, 1.570796, 1.639272],accel_mss,speed_ms,0,blend_radius_m)
    movel([0.068846, -1.395949, -2.563543, -0.752896, 1.570796, 1.639642],accel_mss,speed_ms,0,blend_radius_m)
    movel([0.069096, -1.395864, -2.563605, -0.752919, 1.570796, 1.639893],accel_mss,speed_ms,0,blend_radius_m)
    movel([0.069570, -1.395754, -2.563686, -0.752950, 1.570796, 1.640367],accel_mss,speed_ms,0,blend_radius_m)
    movel([0.070403, -1.395589, -2.563805, -0.752995, 1.570796, 1.641200],accel_mss,speed_ms,0,blend_radius_m)
    movel([0.071125, -1.395481, -2.563884, -0.753024, 1.570796, 1.641922],accel_mss,speed_ms,0,blend_radius_m)
    movel([0.071701, -1.395425, -2.563925, -0.753040, 1.570796, 1.642497],accel_mss,speed_ms,0,blend_radius_m)
    movel([0.071942, -1.395544, -2.563838, -0.753007, 1.570796, 1.642738],accel_mss,speed_ms,0,blend_radius_m)
    movel([0.072038, -1.395800, -2.563652, -0.752937, 1.570796, 1.642834],accel_mss,speed_ms,0,blend_radius_m)
    speed_ms = 0.003
    movel([0.072038, -1.382893, -2.557737, -0.771760, 1.570796, 1.642834],accel_mss,speed_ms,0,blend_radius_m)
    speed_ms = 1.000
    movel([0.072038, -1.358116, -2.545513, -0.808760, 1.570796, 1.642834],accel_mss,speed_ms,0,blend_radius_m)
    movel([0.071087, -1.359327, -2.544680, -0.808382, 1.570796, 1.641883],accel_mss,speed_ms,0,blend_radius_m)
    movel([0.071087, -1.384082, -2.556888, -0.771419, 1.570796, 1.641883],accel_mss,speed_ms,0,blend_radius_m)
    speed_ms = 0.003
    movel([0.071087, -1.393720, -2.561331, -0.757337, 1.570796, 1.641883],accel_mss,speed_ms,0,blend_radius_m)
    speed_ms = 0.007
    movel([0.071759, -1.393816, -2.561262, -0.757311, 1.570796, 1.642556],accel_mss,speed_ms,0,blend_radius_m)
    movel([0.071953, -1.393945, -2.561168, -0.757276, 1.570796, 1.642749],accel_mss,speed_ms,0,blend_radius_m)
    movel([0.072032, -1.394114, -2.561046, -0.757229, 1.570796, 1.642829],accel_mss,speed_ms,0,blend_radius_m)
    movel([0.071840, -1.394423, -2.560821, -0.757144, 1.570796, 1.642637],accel_mss,speed_ms,0,blend_radius_m)
    movel([0.071514, -1.394499, -2.560766, -0.757124, 1.570796, 1.642311],accel_mss,speed_ms,0,blend_radius_m)
    movel([0.071242, -1.394533, -2.560742, -0.757114, 1.570796, 1.642039],accel_mss,speed_ms,0,blend_radius_m)
    movel([0.070950, -1.394556, -2.560725, -0.757108, 1.570796, 1.641746],accel_mss,speed_ms,0,blend_radius_m)
    movel([0.070596, -1.394590, -2.560700, -0.757099, 1.570796, 1.641393],accel_mss,speed_ms,0,blend_radius_m)
    movel([0.070127, -1.394658, -2.560651, -0.757080, 1.570796, 1.640923],accel_mss,speed_ms,0,blend_radius_m)
    movel([0.069629, -1.394746, -2.560587, -0.757056, 1.570796, 1.640426],accel_mss,speed_ms,0,blend_radius_m)
    movel([0.069177, -1.394842, -2.560517, -0.757030, 1.570796, 1.639973],accel_mss,speed_ms,0,blend_radius_m)
    movel([0.068658, -1.394956, -2.560434, -0.756999, 1.570796, 1.639454],accel_mss,speed_ms,0,blend_radius_m)
    movel([0.068335, -1.395002, -2.560401, -0.756986, 1.570796, 1.639131],accel_mss,speed_ms,0,blend_radius_m)
    movel([0.068017, -1.394943, -2.560443, -0.757002, 1.570796, 1.638813],accel_mss,speed_ms,0,blend_radius_m)
    movel([0.068021, -1.394682, -2.560633, -0.757074, 1.570796, 1.638818],accel_mss,speed_ms,0,blend_radius_m)
    movel([0.068685, -1.394201, -2.560983, -0.757205, 1.570796, 1.639482],accel_mss,speed_ms,0,blend_radius_m)
    movel([0.069886, -1.393897, -2.561203, -0.757289, 1.570796, 1.640683],accel_mss,speed_ms,0,blend_radius_m)
    movel([0.071087, -1.393720, -2.561331, -0.757337, 1.570796, 1.641883],accel_mss,speed_ms,0,blend_radius_m)
    speed_ms = 0.003
    movel([0.071087, -1.396977, -2.562796, -0.752617, 1.570796, 1.641883],accel_mss,speed_ms,0,blend_radius_m)
    speed_ms = 0.007
    movel([0.071759, -1.397072, -2.562726, -0.752591, 1.570796, 1.642556],accel_mss,speed_ms,0,blend_radius_m)
    movel([0.071953, -1.397201, -2.562632, -0.752556, 1.570796, 1.642749],accel_mss,speed_ms,0,blend_radius_m)
    movel([0.072032, -1.397369, -2.562509, -0.752510, 1.570796, 1.642829],accel_mss,speed_ms,0,blend_radius_m)
    movel([0.071840, -1.397678, -2.562284, -0.752427, 1.570796, 1.642637],accel_mss,speed_ms,0,blend_radius_m)
    movel([0.071514, -1.397753, -2.562229, -0.752406, 1.570796, 1.642311],accel_mss,speed_ms,0,blend_radius_m)
    movel([0.071242, -1.397787, -2.562205, -0.752397, 1.570796, 1.642039],accel_mss,speed_ms,0,blend_radius_m)
    movel([0.070950, -1.397810, -2.562188, -0.752391, 1.570796, 1.641746],accel_mss,speed_ms,0,blend_radius_m)
    movel([0.070596, -1.397844, -2.562163, -0.752382, 1.570796, 1.641393],accel_mss,speed_ms,0,blend_radius_m)
    movel([0.070127, -1.397911, -2.562114, -0.752364, 1.570796, 1.640923],accel_mss,speed_ms,0,blend_radius_m)
    movel([0.069629, -1.398000, -2.562049, -0.752340, 1.570796, 1.640426],accel_mss,speed_ms,0,blend_radius_m)
    movel([0.069177, -1.398096, -2.561979, -0.752314, 1.570796, 1.639973],accel_mss,speed_ms,0,blend_radius_m)
    movel([0.068658, -1.398209, -2.561896, -0.752283, 1.570796, 1.639454],accel_mss,speed_ms,0,blend_radius_m)
    movel([0.068335, -1.398255, -2.561863, -0.752271, 1.570796, 1.639131],accel_mss,speed_ms,0,blend_radius_m)
    movel([0.068017, -1.398196, -2.561906, -0.752287, 1.570796, 1.638813],accel_mss,speed_ms,0,blend_radius_m)
    movel([0.068021, -1.397936, -2.562096, -0.752357, 1.570796, 1.638818],accel_mss,speed_ms,0,blend_radius_m)
    movel([0.068685, -1.397456, -2.562446, -0.752487, 1.570796, 1.639482],accel_mss,speed_ms,0,blend_radius_m)
    movel([0.069886, -1.397153, -2.562667, -0.752569, 1.570796, 1.640683],accel_mss,speed_ms,0,blend_radius_m)
    movel([0.071087, -1.396977, -2.562796, -0.752617, 1.570796, 1.641883],accel_mss,speed_ms,0,blend_radius_m)
    speed_ms = 0.003
    movel([0.071087, -1.384082, -2.556888, -0.771419, 1.570796, 1.641883],accel_mss,speed_ms,0,blend_radius_m)
    speed_ms = 1.000
    movel([0.071087, -1.359327, -2.544680, -0.808382, 1.570796, 1.641883],accel_mss,speed_ms,0,blend_radius_m)
    movel([0.070689, -1.360858, -2.543624, -0.807908, 1.570796, 1.641485],accel_mss,speed_ms,0,blend_radius_m)
    movel([0.070689, -1.385584, -2.555813, -0.770992, 1.570796, 1.641485],accel_mss,speed_ms,0,blend_radius_m)
    speed_ms = 0.003
    movel([0.070689, -1.395211, -2.560249, -0.756929, 1.570796, 1.641485],accel_mss,speed_ms,0,blend_radius_m)
    speed_ms = 0.007
    movel([0.071288, -1.395336, -2.560158, -0.756895, 1.570796, 1.642084],accel_mss,speed_ms,0,blend_radius_m)
    movel([0.071443, -1.395487, -2.560048, -0.756854, 1.570796, 1.642240],accel_mss,speed_ms,0,blend_radius_m)
    movel([0.071331, -1.395822, -2.559804, -0.756763, 1.570796, 1.642128],accel_mss,speed_ms,0,blend_radius_m)
    movel([0.070938, -1.395963, -2.559701, -0.756724, 1.570796, 1.641734],accel_mss,speed_ms,0,blend_radius_m)
    movel([0.070676, -1.396000, -2.559674, -0.756714, 1.570796, 1.641472],accel_mss,speed_ms,0,blend_radius_m)
    movel([0.070376, -1.396032, -2.559651, -0.756706, 1.570796, 1.641172],accel_mss,speed_ms,0,blend_radius_m)
    movel([0.070079, -1.396055, -2.559635, -0.756699, 1.570796, 1.640875],accel_mss,speed_ms,0,blend_radius_m)
    movel([0.069755, -1.396088, -2.559611, -0.756691, 1.570796, 1.640551],accel_mss,speed_ms,0,blend_radius_m)
    movel([0.069368, -1.396148, -2.559567, -0.756674, 1.570796, 1.640165],accel_mss,speed_ms,0,blend_radius_m)
    movel([0.068988, -1.396224, -2.559511, -0.756654, 1.570796, 1.639784],accel_mss,speed_ms,0,blend_radius_m)
    movel([0.068671, -1.396306, -2.559452, -0.756631, 1.570796, 1.639468],accel_mss,speed_ms,0,blend_radius_m)
    movel([0.068109, -1.396441, -2.559353, -0.756595, 1.570796, 1.638905],accel_mss,speed_ms,0,blend_radius_m)
    movel([0.067804, -1.396414, -2.559373, -0.756602, 1.570796, 1.638600],accel_mss,speed_ms,0,blend_radius_m)
    movel([0.067930, -1.395974, -2.559694, -0.756722, 1.570796, 1.638726],accel_mss,speed_ms,0,blend_radius_m)
    movel([0.068477, -1.395624, -2.559948, -0.756817, 1.570796, 1.639273],accel_mss,speed_ms,0,blend_radius_m)
    movel([0.069587, -1.395350, -2.560147, -0.756891, 1.570796, 1.640383],accel_mss,speed_ms,0,blend_radius_m)
    movel([0.070689, -1.395211, -2.560249, -0.756929, 1.570796, 1.641485],accel_mss,speed_ms,0,blend_radius_m)
    speed_ms = 0.003
    movel([0.070689, -1.398463, -2.561711, -0.752215, 1.570796, 1.641485],accel_mss,speed_ms,0,blend_radius_m)
    speed_ms = 0.007
    movel([0.071288, -1.398588, -2.561619, -0.752182, 1.570796, 1.642084],accel_mss,speed_ms,0,blend_radius_m)
    movel([0.071443, -1.398738, -2.561510, -0.752141, 1.570796, 1.642240],accel_mss,speed_ms,0,blend_radius_m)
    movel([0.071331, -1.399073, -2.561265, -0.752051, 1.570796, 1.642128],accel_mss,speed_ms,0,blend_radius_m)
    movel([0.070938, -1.399214, -2.561162, -0.752014, 1.570796, 1.641734],accel_mss,speed_ms,0,blend_radius_m)
    movel([0.070676, -1.399250, -2.561135, -0.752004, 1.570796, 1.641472],accel_mss,speed_ms,0,blend_radius_m)
    movel([0.070376, -1.399282, -2.561112, -0.751995, 1.570796, 1.641172],accel_mss,speed_ms,0,blend_radius_m)
    movel([0.070079, -1.399305, -2.561095, -0.751989, 1.570796, 1.640875],accel_mss,speed_ms,0,blend_radius_m)
    movel([0.069755, -1.399338, -2.561071, -0.751980, 1.570796, 1.640551],accel_mss,speed_ms,0,blend_radius_m)
    movel([0.069368, -1.399397, -2.561027, -0.751964, 1.570796, 1.640165],accel_mss,speed_ms,0,blend_radius_m)
    movel([0.068988, -1.399473, -2.560972, -0.751944, 1.570796, 1.639784],accel_mss,speed_ms,0,blend_radius_m)
    movel([0.068671, -1.399555, -2.560912, -0.751922, 1.570796, 1.639468],accel_mss,speed_ms,0,blend_radius_m)
    movel([0.068109, -1.399690, -2.560813, -0.751886, 1.570796, 1.638905],accel_mss,speed_ms,0,blend_radius_m)
    movel([0.067804, -1.399663, -2.560833, -0.751893, 1.570796, 1.638600],accel_mss,speed_ms,0,blend_radius_m)
    movel([0.067930, -1.399224, -2.561154, -0.752011, 1.570796, 1.638726],accel_mss,speed_ms,0,blend_radius_m)
    movel([0.068477, -1.398875, -2.561409, -0.752104, 1.570796, 1.639273],accel_mss,speed_ms,0,blend_radius_m)
    movel([0.069587, -1.398602, -2.561609, -0.752178, 1.570796, 1.640383],accel_mss,speed_ms,0,blend_radius_m)
    movel([0.070689, -1.398463, -2.561711, -0.752215, 1.570796, 1.641485],accel_mss,speed_ms,0,blend_radius_m)
    speed_ms = 0.003
    movel([0.070689, -1.385584, -2.555813, -0.770992, 1.570796, 1.641485],accel_mss,speed_ms,0,blend_radius_m)
    speed_ms = 1.000
    movel([0.070689, -1.360858, -2.543624, -0.807908, 1.570796, 1.641485],accel_mss,speed_ms,0,blend_radius_m)
    movel([0.069782, -1.362641, -2.542390, -0.807359, 1.570796, 1.640579],accel_mss,speed_ms,0,blend_radius_m)
    movel([0.069782, -1.387335, -2.554556, -0.770498, 1.570796, 1.640579],accel_mss,speed_ms,0,blend_radius_m)
    speed_ms = 0.003
    movel([0.069782, -1.396948, -2.558984, -0.756458, 1.570796, 1.640579],accel_mss,speed_ms,0,blend_radius_m)
    speed_ms = 0.007
    movel([0.070081, -1.397018, -2.558932, -0.756439, 1.570796, 1.640877],accel_mss,speed_ms,0,blend_radius_m)
    movel([0.070082, -1.397273, -2.558746, -0.756370, 1.570796, 1.640878],accel_mss,speed_ms,0,blend_radius_m)
    movel([0.069829, -1.397430, -2.558632, -0.756328, 1.570796, 1.640625],accel_mss,speed_ms,0,blend_radius_m)
    movel([0.069576, -1.397509, -2.558574, -0.756306, 1.570796, 1.640372],accel_mss,speed_ms,0,blend_radius_m)
    movel([0.069100, -1.397609, -2.558501, -0.756279, 1.570796, 1.639897],accel_mss,speed_ms,0,blend_radius_m)
    movel([0.068697, -1.397625, -2.558489, -0.756275, 1.570796, 1.639493],accel_mss,speed_ms,0,blend_radius_m)
    movel([0.068424, -1.397557, -2.558538, -0.756293, 1.570796, 1.639220],accel_mss,speed_ms,0,blend_radius_m)
    movel([0.068377, -1.397306, -2.558722, -0.756361, 1.570796, 1.639174],accel_mss,speed_ms,0,blend_radius_m)
    movel([0.068857, -1.397068, -2.558896, -0.756425, 1.570796, 1.639653],accel_mss,speed_ms,0,blend_radius_m)
    movel([0.069345, -1.396961, -2.558974, -0.756454, 1.570796, 1.640141],accel_mss,speed_ms,0,blend_radius_m)
    movel([0.069782, -1.396948, -2.558984, -0.756458, 1.570796, 1.640579],accel_mss,speed_ms,0,blend_radius_m)
    speed_ms = 0.003
    movel([0.069782, -1.400195, -2.560443, -0.751751, 1.570796, 1.640579],accel_mss,speed_ms,0,blend_radius_m)
    speed_ms = 0.007
    movel([0.070081, -1.400265, -2.560391, -0.751733, 1.570796, 1.640877],accel_mss,speed_ms,0,blend_radius_m)
    movel([0.070082, -1.400520, -2.560205, -0.751665, 1.570796, 1.640878],accel_mss,speed_ms,0,blend_radius_m)
    movel([0.069829, -1.400676, -2.560090, -0.751623, 1.570796, 1.640625],accel_mss,speed_ms,0,blend_radius_m)
    movel([0.069576, -1.400755, -2.560032, -0.751602, 1.570796, 1.640372],accel_mss,speed_ms,0,blend_radius_m)
    movel([0.069100, -1.400855, -2.559959, -0.751576, 1.570796, 1.639897],accel_mss,speed_ms,0,blend_radius_m)
    movel([0.068697, -1.400871, -2.559947, -0.751571, 1.570796, 1.639493],accel_mss,speed_ms,0,blend_radius_m)
    movel([0.068424, -1.400803, -2.559996, -0.751589, 1.570796, 1.639220],accel_mss,speed_ms,0,blend_radius_m)
    movel([0.068377, -1.400553, -2.560180, -0.751656, 1.570796, 1.639174],accel_mss,speed_ms,0,blend_radius_m)
    movel([0.068857, -1.400315, -2.560355, -0.751719, 1.570796, 1.639653],accel_mss,speed_ms,0,blend_radius_m)
    movel([0.069345, -1.400209, -2.560433, -0.751748, 1.570796, 1.640141],accel_mss,speed_ms,0,blend_radius_m)
    movel([0.069782, -1.400195, -2.560443, -0.751751, 1.570796, 1.640579],accel_mss,speed_ms,0,blend_radius_m)
    speed_ms = 0.003
    movel([0.069782, -1.387335, -2.554556, -0.770498, 1.570796, 1.640579],accel_mss,speed_ms,0,blend_radius_m)
    speed_ms = 1.000
    movel([0.069782, -1.362641, -2.542390, -0.807359, 1.570796, 1.640579],accel_mss,speed_ms,0,blend_radius_m)
    movel([0.070729, -1.364236, -2.541282, -0.806871, 1.570796, 1.641526],accel_mss,speed_ms,0,blend_radius_m)
    movel([0.070729, -1.388900, -2.553429, -0.770060, 1.570796, 1.641526],accel_mss,speed_ms,0,blend_radius_m)
    speed_ms = 0.003
